(* CODESYS project Cowbell_Tracy_rev_2.project

Project tree, tasks and I/O mapping:
  Device : PAC320-CXX2X-XX, Parker Hannifin, order no. PAC320-CXX2X-XX, version 3.5.5.20
    application Application
      libraries: Util, 3.5.1.0 (System); CAA Types Extern, 3.5.5.0 (CAA Technical Workgroup); SysTypes Interfaces, * (System); CmpIecTask, 3.5.5.0 (System); SysFile, 3.5.5.0 (System); CmpErrors Interfaces, * (System); Unit Conversion Interfaces, * (Intern); SysTime, 3.5.5.0 (System)
      task EtherCAT_Master (externalevent, external event EVENT_ECM_DC, priority 0) calls EtherCAT_Master.EtherCAT_Task [EtherCAT_Master.EtherCAT_Task], DC_Monitor, RunLights, Rungs_First_500, Rungs_Second_500, RunMotion_All, Recovery, LogHiCycleCount
      task Slow_Task (cyclic, interval t#150ms, priority 20) calls PLC_PRG_1, Run_FileCopy, LogData
      global variables GVL
      global variables PersistentVars
      SymbolConfiguration
    SoftMotion General Axis Pool
      ZZ : SM_Drive_Virtual, 3S - Smart Software Solutions GmbH, order no. 1805, version 3.5.5.0
          settings: fRampJerk = 1e7
      A : SM_Drive_Virtual, 3S - Smart Software Solutions GmbH, order no. 1805, version 3.5.5.0
          settings: fRampJerk = 1e7
    EtherCAT_Master : PAC320 EtherCAT Master, Parker Hannifin, order no. PAC320-XXXXX-XX, version 3.5.5.0
        settings: MasterCycleTime = 1000
      Accelnet : Accelnet EtherCAT Drive (CoE) SoftMotion, Copley Controls Corp., version 3.5.5.0
          settings: EnableExpertSettings = True; StationAlias = 16; Optional = True; DC sync0 cycletime = 500; DC sync0 factor = 'x 1'; DC sync0 shift time = 0; DC sync1 cycletime = 500; DC sync1 factor = 'x 1'; DC sync1 shift time = 0; DCSetting = -1
          unmapped channels: Control word, Modes of operation, Target Position, Status word, Modes of operation display, Actual position
        Y : SM_Drive_ETC_Copley, 3S - Smart Software Solutions GmbH, order no. 0, version 3.5.5.0
            settings: AddressOffset_8010 = 20; BitOffset_8010 = 0; BitLength_8010 = 16; Address_8010 = '%QW10'; Type_8010 = 'UINT'; AddressPointer_8010 = ADR(%QW10); AddressOffset_8020 = 22; BitOffset_8020 = 0; BitLength_8020 = 8; Address_8020 = '%QB22'; Type_8020 = 'USINT'; AddressPointer_8020 = ADR(%QB22); AddressOffset_8030 = 24; BitOffset_8030 = 0; BitLength_8030 = 32; Address_8030 = '%QD6'; Type_8030 = 'DINT'; AddressPointer_8030 = ADR(%QD6); AddressOffset_8040 = 16#FFFFFFFF; BitOffset_8040 = 0; BitLength_8040 = 0; Address_8040 = ''; Type_8040 = ''; AddressPointer_8040 = 0; AddressOffset_8050 = 16#FFFFFFFF; BitOffset_8050 = 0; BitLength_8050 = 0; Address_8050 = ''; Type_8050 = ''; AddressPointer_8050 = 0; AdrOffset_8060 = 16#FFFFFFFF; BitOffset_8060 = 0; BitLength_8060 = 0; Address_8060 = ''; Type_8060 = ''; AddressPointer_8060 = 0; AdrOffset_8070 = 16#FFFFFFFF; BitOffset_8070 = 0; BitLength_8070 = 0; Address_8070 = '';
              Type_8070 = ''; AddressPointer_8070 = 0; AddressOffset_8510 = 24; BitOffset_8510 = 0; BitLength_8510 = 16; Address_8510 = '%IW12'; Type_8510 = 'UINT'; AddressPointer_8510 = ADR(%IW12); AddressOffset_8520 = 26; BitOffset_8520 = 0; BitLength_8520 = 8; Address_8520 = '%IB26'; Type_8520 = 'USINT'; AddressPointer_8520 = ADR(%IB26); AddressOffset_8530 = 28; BitOffset_8530 = 0; BitLength_8530 = 32; Address_8530 = '%ID7'; Type_8530 = 'DINT'; AddressPointer_8530 = ADR(%ID7); AddressOffset_8540 = 16#FFFFFFFF; BitOffset_8540 = 0; BitLength_8540 = 0; Address_8540 = ''; Type_8540 = ''; AddressPointer_8540 = 0; AddressOffset_8550 = 16#FFFFFFFF; BitOffset_8550 = 0; BitLength_8550 = 0; Address_8550 = ''; Type_8550 = ''; AddressPointer_8550 = 0
      Xenus_Plus_XEL : Xenus Plus EtherCAT Drive (CoE), Copley Controls, version Revision=16#00010003
          settings: EnableExpertSettings = True; Watchdog register 0400 = 2498; Watchdog register 0410 = 1000; Watchdog register 0420 = 1000; StationAlias = 17; DC sync0 cycletime = 1000; DC enable = 1; DC sync0 enable = 1; DC sync0 factor = 'x 1'; DC sync0 shift time = 0; DC sync1 cycletime = 1000; DC sync1 factor = 'x 1'; DC sync1 shift time = 0; DCSetting = 0; DC cyclic unit control = 48
          unmapped channels: Control word, Profile target position, Velocity offset, Torque offset, Status word, Actual motor position, Position loop error., Actual motor velocity, Torque actual value
        X : SM_Drive_ETC_GenericDSP402, 3S - Smart Software Solutions GmbH, order no. 0, version 3.5.5.0
            settings: dwRatioTechUnitsDenom = 4000; fPositionPeriod = 1; fRampJerk = 1e7; fSWLimitDeceleration = 0.0; fSWErrorMaxDistance = 0.0; ScalingIncs = 4000; AdrOffset_8010 = 4; BitOffset_8010 = 0; BitLength_8010 = 16; Address_8010 = '%QW2'; Type_8010 = 'UINT'; AddressPointer_8010 = ADR(%QW2); AdrOffset_8020 = 8; BitOffset_8020 = 0; BitLength_8020 = 32; Address_8020 = '%QD2'; Type_8020 = 'DINT'; AddressPointer_8020 = ADR(%QD2); AdrOffset_8030 = 16#FFFFFFFF; BitOffset_8030 = 0; BitLength_8030 = 0; Address_8030 = ''; Type_8030 = ''; AddressPointer_8030 = 0; AdrOffset_8040 = 16#FFFFFFFF; BitOffset_8040 = 0; BitLength_8040 = 0; Address_8040 = ''; Type_8040 = ''; AddressPointer_8040 = 0; AdrOffset_8050 = 16#FFFFFFFF; BitOffset_8050 = 0; BitLength_8050 = 0; Address_8050 = ''; Type_8050 = ''; AddressPointer_8050 = 0; AdrOffset_8060 = 16#FFFFFFFF; BitOffset_8060 = 0; BitLength_8060 = 0; Address_8060 = '';
              Type_8060 = ''; AddressPointer_8060 = 0; AdrOffset_8070 = 12; BitOffset_8070 = 0; BitLength_8070 = 32; Address_8070 = '%QD3'; Type_8070 = 'DINT'; AddressPointer_8070 = ADR(%QD3); AdrOffset_8080 = 16; BitOffset_8080 = 0; BitLength_8080 = 16; Address_8080 = '%QW8'; Type_8080 = 'INT'; AddressPointer_8080 = ADR(%QW8); AdrOffset_8510 = 4; BitOffset_8510 = 0; BitLength_8510 = 16; Address_8510 = '%IW2'; Type_8510 = 'UINT'; AddressPointer_8510 = ADR(%IW2); AdrOffset_8520 = 8; BitOffset_8520 = 0; BitLength_8520 = 32; Address_8520 = '%ID2'; Type_8520 = 'DINT'; AddressPointer_8520 = ADR(%ID2); AdrOffset_8530 = 16; BitOffset_8530 = 0; BitLength_8530 = 32; Address_8530 = '%ID4'; Type_8530 = 'DINT'; AddressPointer_8530 = ADR(%ID4); AdrOffset_8540 = 20; BitOffset_8540 = 0; BitLength_8540 = 16; Address_8540 = '%IW10'; Type_8540 = 'INT'; AddressPointer_8540 = ADR(%IW10); AdrOffset_8550 = 16#FFFFFFFF; BitOffset_8550 = 0;
              BitLength_8550 = 0; Address_8550 = ''; Type_8550 = ''; AddressPointer_8550 = 0; AdrOffset_8560 = 16#FFFFFFFF; BitOffset_8560 = 0; BitLength_8560 = 0; Address_8560 = ''; Type_8560 = ''; AddressPointer_8560 = 0; AdrOffset_8570 = 16#FFFFFFFF; BitOffset_8570 = 0; BitLength_8570 = 0; Address_8570 = ''; Type_8570 = ''; AddressPointer_8570 = 0; AdrOffset_8580 = 16#FFFFFFFF; BitOffset_8580 = 0; BitLength_8580 = 0; Address_8580 = ''; Type_8580 = ''; AddressPointer_8580 = 0; AdrOffset_8590 = 16#FFFFFFFF; BitOffset_8590 = 0; BitLength_8590 = 0; Address_8590 = ''; Type_8590 = ''; AddressPointer_8590 = 0; AdrOffset_8600 = 16#FFFFFFFF; BitOffset_8600 = 0; BitLength_8600 = 0; Address_8600 = ''; Type_8600 = ''; AddressPointer_8600 = 0; AdrOffset_8600 = 16#FFFFFFFF; BitOffset_8600 = 0; BitLength_8600 = 0; Address_8610 = ''; Type_8610 = ''; AddressPointer_8610 = 0
      PAC320_BusCoupler : PAC320 BusCoupler, Parker Hannifin, version Revision=16#00000001
          settings: EnableExpertSettings = True; StationAlias = 1; DC sync0 cycletime = 500; DC enable = 1; DC sync0 enable = 1; DC sync0 factor = 'x 1'; DC sync0 shift time = 0; DC sync1 cycletime = 500; DC sync1 enable = 0; DC sync1 factor = 'x 1'; DC sync1 shift time = 0
        PACIO_DI16_DO16 : DI16/DO16 1ms 0.5A (PACIO-450-03), Parker Hannifin, version Revision=16#00000001
            settings: StationAlias = 0; DC sync0 cycletime = 500; DC sync1 cycletime = 500
            output A_Output00 : BIT  // DigitalOutput0
            output A_Output01 : BIT  // DigitalOutput1
            output A_Output02 : BIT  // DigitalOutput2
            output A_Output03 : BIT  // DigitalOutput3
            output A_Output04 : BIT  // DigitalOutput4
            output A_Output05 : BIT  // DigitalOutput5
            output A_Output06 : BIT  // DigitalOutput6
            output A_Output07 : BIT  // DigitalOutput7
            output A_Output08 : BIT  // DigitalOutput8
            output A_Output09 : BIT  // DigitalOutput9
            output A_Output10 : BIT  // DigitalOutput10
            output A_Output11 : BIT  // DigitalOutput11
            output A_Output12 : BIT  // DigitalOutput12
            output A_Output13 : BIT  // DigitalOutput13
            output A_Output14 : BIT  // DigitalOutput14
            output A_Output15 : BIT  // DigitalOutput15
            input  A_Input00 : BIT  // DigitalInput0
            input  A_Input01 : BIT  // DigitalInput1
            input  A_Input02 : BIT  // DigitalInput2
            input  A_Input03 : BIT  // DigitalInput3
            input  A_Input04 : BIT  // DigitalInput4
            input  A_Input05 : BIT  // DigitalInput5
            input  A_Input06 : BIT  // DigitalInput6
            input  A_Input07 : BIT  // DigitalInput7
            input  In_Power : BIT  // DigitalInput8
            input  In_Reset : BIT  // DigitalInput9
            input  In_Neg : BIT  // DigitalInput10
            input  In_Pos : BIT  // DigitalInput11
            input  In_Zero : BIT  // DigitalInput12
            input  In_Start : BIT  // DigitalInput13
            input  In_Stop : BIT  // DigitalInput14
            input  In_Cycle : BIT  // DigitalInput15
        PACIO_DI16_DO16_1 : DI16/DO16 1ms 0.5A (PACIO-450-03), Parker Hannifin, version Revision=16#00000001
            settings: StationAlias = 0; DC sync0 cycletime = 500; DC sync1 cycletime = 500
            output B_Output00 : BIT  // DigitalOutput0
            output B_Output01 : BIT  // DigitalOutput1
            output B_Output02 : BIT  // DigitalOutput2
            output B_Output03 : BIT  // DigitalOutput3
            output B_Output04 : BIT  // DigitalOutput4
            output B_Output05 : BIT  // DigitalOutput5
            output B_Output06 : BIT  // DigitalOutput6
            output B_Output07 : BIT  // DigitalOutput7
            output B_Output08 : BIT  // DigitalOutput8
            output B_Output09 : BIT  // DigitalOutput9
            output B_Output10 : BIT  // DigitalOutput10
            output B_Output11 : BIT  // DigitalOutput11
            output B_Output12 : BIT  // DigitalOutput12
            output B_Output13 : BIT  // DigitalOutput13
            output B_Output14 : BIT  // DigitalOutput14
            output B_Output15 : BIT  // DigitalOutput15
            input  B_Input00 : BIT  // DigitalInput0
            input  B_Input01 : BIT  // DigitalInput1
            input  B_Input02 : BIT  // DigitalInput2
            input  B_Input03 : BIT  // DigitalInput3
            input  B_Input04 : BIT  // DigitalInput4
            input  B_Input05 : BIT  // DigitalInput5
            input  B_Input06 : BIT  // DigitalInput6
            input  B_Input07 : BIT  // DigitalInput7
            input  B_Input08 : BIT  // DigitalInput8
            input  B_Input09 : BIT  // DigitalInput9
            input  B_Input10 : BIT  // DigitalInput10
            input  B_Input11 : BIT  // DigitalInput11
            input  B_Input12 : BIT  // DigitalInput12
            input  B_Input13 : BIT  // DigitalInput13
            input  B_Input14 : BIT  // DigitalInput14
            input  B_Input15 : BIT  // DigitalInput15
      Compax3_EtherCat_DS402_CoE : C3SxxxVxFxxI31T11Mxx_OpMode08 V2.05 SoftMotion, Parker Hannifin, version 3.5.5.0
          settings: EnableExpertSettings = True; StationAlias = 1006; Optional = True; DC sync0 cycletime = 4000; DC enable = 1; DC sync0 enable = 1; DC sync0 factor = 'x 4'; DC sync0 shift time = 0; DC sync1 cycletime = 4000; DC sync1 enable = 0; DC sync1 shift time = 0
          unmapped channels: Controlword, Target Position, Dig.Outputs, ModeofOperation, Statusword, Actual Position, Dig.Inputs, ModeOfOperationDisplay
        Z : SM_Drive_ETC_PARKER, 3S - Smart Software Solutions GmbH, order no. 0, version 3.5.5.0
            settings: dwRatioTechUnitsDenom = 4096; ScalingIncs = 4096; AdrOffset_8010 = 28; BitOffset_8010 = 0; BitLength_8010 = 16; Address_8010 = '%QW14'; Type_8010 = 'UINT'; AddressPointer_8010 = ADR(%QW14); AdrOffset_8020 = 32; BitOffset_8020 = 0; BitLength_8020 = 32; Address_8020 = '%QD8'; Type_8020 = 'DINT'; AddressPointer_8020 = ADR(%QD8); AdrOffset_8030 = 38; BitOffset_8030 = 0; BitLength_8030 = 16; Address_8030 = '%QW19'; Type_8030 = 'INT'; AddressPointer_8030 = ADR(%QW19); AdrOffset_8040 = 36; BitOffset_8040 = 0; BitLength_8040 = 16; Address_8040 = '%QW18'; Type_8040 = 'UINT'; AddressPointer_8040 = ADR(%QW18); AdrOffset_8510 = 32; BitOffset_8510 = 0; BitLength_8510 = 16; Address_8510 = '%IW16'; Type_8510 = 'UINT'; AddressPointer_8510 = ADR(%IW16); AdrOffset_8520 = 16#FFFFFFFF; BitOffset_8520 = 0; BitLength_8520 = 0; Address_8520 = ''; Type_8520 = ''; AddressPointer_8520 = 0; AdrOffset_8530 = 42; BitOffset_8530 = 0;
              BitLength_8530 = 16; Address_8530 = '%IW21'; Type_8530 = 'INT'; AddressPointer_8530 = ADR(%IW21); AdrOffset_8540 = 40; BitOffset_8540 = 0; BitLength_8540 = 16; Address_8540 = '%IW20'; Type_8540 = 'UINT'; AddressPointer_8540 = ADR(%IW20); AdrOffset_8550 = 36; BitOffset_8550 = 0; BitLength_8550 = 32; Address_8550 = '%ID9'; Type_8550 = 'DINT'; AddressPointer_8550 = ADR(%ID9)
    Ethernet : Ethernet, 3S - Smart Software Solutions GmbH, version 3.4.2.0
      ModbusTCP_Slave_Device : ModbusTCP Slave Device, 3S - Smart Software Solutions GmbH, version 3.5.5.0
          input  Application.DC_Monitor.HMI_ResetCounter : WORD  // Inputs.Inputs
          output Application.DC_Monitor.Captured_CycleTime_Avg : WORD  // Outputs.Outputs
          output Application.DC_Monitor.Captured_CycleTime_Max : WORD  // Outputs.Outputs
          output Application.DC_Monitor.Captured_CycleTime_Min : WORD  // Outputs.Outputs
          output Application.DC_Monitor.Captured_MaxTotalSyncBufferAvg : WORD  // Outputs.Outputs
          output Application.DC_Monitor.CycleTime_Avg : WORD  // Outputs.Outputs
          output Application.DC_Monitor.CycleTime_Max : WORD  // Outputs.Outputs
          output Application.DC_Monitor.CycleTime_Min : WORD  // Outputs.Outputs
          output Application.DC_Monitor.CycleTime_Count : WORD  // Outputs.Outputs
          output Application.DC_Monitor.CycleTime_Last : WORD  // Outputs.Outputs
          output Application.MaxTotalSyncBufferAvg : WORD  // Outputs.Outputs
          output Application.DC_Monitor.TotalSyncBufferAvg : WORD  // Outputs.Outputs
          output Application.RunLights.iCycle : WORD  // Outputs.Outputs
          output Application.RunMotion_All.DoMotion_X.HMI_ActualPosition : WORD  // Outputs.Outputs
          output Application.DC_Monitor.HMI_DC_InSync : WORD  // Outputs.Outputs
          output Application.dcWindow : WORD  // Outputs.Outputs
          output Application.gSyncErrors : WORD  // Outputs.Outputs
          unmapped channels: Inputs, Outputs
  program PLC_PRG [CFC]
  program RunSDO_AOut [ST]
  function block GetSDO_AOut [CFC]
  function block GetSDO [CFC]
  function block SetOutputs [ST]
  function block GetInputs [ST]
  function block SetAnalogVoltage [ST]
  function VOLTS_to_UINT [ST]
  function UINT_to_VOLTS [ST]
  program RunSDO [ST]
  function block GetAnalogVoltage [ST]
  function block InitSDO [ST]
  function block ConfigAnalogVoltage [ST]
  program RunMotion_old [ST]
  function block IO_AxisControl [CFC]
  program POU_X [CFC]
  function block SetSDO_AOut [CFC]
  function block InitSDO_Y [ST]
  program RunMotion_Y_old [ST]
  program RunSDO_Y [ST]
  program RunSDO_AOut_Y [ST]
  function block GetSDO_Y [CFC]
  function block GetSDO_AOut_Y [CFC]
  function block SetSDO_AOut_Y [CFC]
  function GetHeaderString [ST]
  program DC_Monitor [ST]
  program RunLights [ST]
  program RunMotion_Z_old [ST]
  program RunMotion_A [ST]
  function block MotionFB [ST]
  program Recovery [ST]
  program RunMotion_All [ST]
  function GetLogMsgString [ST]
  program LogHiCycleCount [ST]
  function GetTimeStampString [ST]
  text list GlobalTextList
  function AllTaskInfo [ST]
  function CurrentTaskInfo [ST]
  function ResetTaskInfo [ST]
  program Rungs_First_500 [LD]
  program Rungs_Second_500 [LD]
  program RunMotion [ST]
  program RunMotion_Y [ST]
  program RunMotion_Z [ST]
  function block Test_FileCopy [ST]
  program Run_FileCopy [CFC]
  program PLC_PRG_1 [ST]
  program LogData [ST]
  function My_FLOAT_TO_STRING [ST]
  function GetTimeStampString_1 [ST]
*)

// Device/Application/GVL
VAR_GLOBAL
	g_PosDistance:REAL := 20.0;
	g_NegDistance:REAL := -20.0;
	g_Vel:REAL := 5.0;
	g_Acc:REAL := 10.0;
	//In_Power : BOOL ;
	//In_Reset : BOOL;
	//In_Pos : BOOL;
	//In_Neg : BOOL;
	//In_Stop : BOOL;
	//In_Zero : BOOL;
	g_MoveDwellPos : BOOL := FALSE;
	g_MoveDwellNeg : BOOL := FALSE;
	g_MoveDwellPos_Y : BOOL := FALSE;
	g_MoveDwellNeg_Y : BOOL := FALSE;
	g_MoveDwellPos_Z : BOOL := FALSE;
	g_MoveDwellNeg_Z : BOOL := FALSE;
	g_MoveDwellPos_A : BOOL := FALSE;
	g_MoveDwellNeg_A : BOOL := FALSE;
	g_GotSDO_PostionPos : BOOL;
	g_GotSDO_PostionNeg : BOOL;
	g_GotSDO_Y_PostionPos : BOOL;
	g_GotSDO_Y_PostionNeg : BOOL;
	DC_InSync: BOOL;
	g_FirstSync: BOOL;
	g_LostSync: BOOL;
	
	
	//ScanTimeMax: DINT;
	//ScanTimeMin: DINT;
	//dcWindow: WORD := 50;

	//MaxScanTime: DINT;
	//MaxSyncTime: DINT;
	//MinSyncTime: DINT;
	//MaxTotalSyncBufferAvg: DINT;
	MyArray: ARRAY[0..9, 0..9] OF REAL;
END_VAR

// Device/Application/PersistentVars
VAR_GLOBAL PERSISTENT RETAIN
	ScanTimeMax: DINT;
	ScanTimeMin: DINT;
	dcWindow: WORD ;

	MaxScanTime: DINT;
	MaxSyncTime: DINT;
	MinSyncTime: DINT;
	MaxTotalSyncBufferAvg: DINT;

	gSyncErrors: DINT;
END_VAR

// DC_Monitor
PROGRAM DC_Monitor
VAR
	TurnON_LED_A: BOOL;
	TurnON_LED_B: BOOL;
	m_master: INT;
	ResetLED: BOOL := FALSE;
	iLoopCount: UINT;
	CurrentScanTime: DINT;
	CurrentSyncTime: DINT;
	SyncBufferMax: DINT;
	TotalSyncBuffer: DINT;
	TotalSyncBufferAvg: DINT;
	tTask 			: Task_Info2; (* Information about the task *)
	pTask2			: POINTER  TO Task_Info2;
	aIecTasks 		: ARRAY[1..20] OF Task_Info2; (* Information about all tasks *)
	sAppName		: STRING := 'Application';
	
	hCurrentTask	: RTS_IEC_HANDLE; (* Current task *)
	hSlowTask		: RTS_IEC_HANDLE; (* The slower task handle*)
	hReloaded 		: RTS_IEC_HANDLE; (* Reloaded task *)
	Result			: RTS_IEC_RESULT; (* Result Code *)
	ResetStats : BOOL;
	ResetResult		: RTS_IEC_RESULT; (* Reset Result Code *)
	DoReset : BOOL := FALSE;
	DoAutoReset : BOOL := FALSE;
	Capture_Done : BOOL := FALSE;
	Captured_CycleTime_Avg : DWORD := 0;
	Captured_CycleTime_Max : DWORD := 0;
	Captured_CycleTime_Min : DWORD := 0;
	Captured_MaxTotalSyncBufferAvg : DINT := 0;
	
	
	CyclesIn5min: UDINT;
	CycleTime_Avg: DWORD;
	CycleTime_Max: DWORD;
	CycleTime_Min: DWORD;
	CycleTime_Last: DWORD;
	CycleTime_Count: DWORD;
	
	HMI_ResetCounter : WORD;
	HMI_DC_InSync : WORD;
	
END_VAR

EtherCAT_Master();
dcWindow := EtherCAT_Master.DCInSyncWindow;
//ScanTimeMax := EtherCAT_Master.m_master.m_diMaxSyncTime;
//ScanTimeMin := EtherCAT_Master.m_master.m_diMinSyncTime;
DC_InSync := EtherCAT_Master.xDistributedClockInSync;
(* Current task information, some of these information can be find in the Task Configuration under the monitor tab.*)
tTask := CurrentTaskInfo();
	CycleTime_Avg := tTask.dwAverageCycleTime;
	CycleTime_Max := tTask.dwMaxCycleTime;
	CycleTime_Min := tTask.dwMinCycleTime;
	CycleTime_Last := tTask.dwCycleTime; 
	CycleTime_Count := tTask.dwCycleCount / 2000;
	DoReset := HMI_ResetCounter.0;
	HMI_DC_InSync.0 := DC_InSync;
	

IF DoReset OR DoAutoReset THEN
	ResetResult := ResetTaskInfo();
	MaxTotalSyncBufferAvg := 0;
	Capture_Done := FALSE;
	Captured_CycleTime_Avg := 0;
	Captured_CycleTime_Max := 0;
	Captured_CycleTime_Min := 0;
	Captured_MaxTotalSyncBufferAvg := 0;
	DoReset := FALSE;
	DoAutoReset := FALSE;
END_IF;


TotalSyncBuffer := 0;
FOR iLoopCount:=0 TO ETHERCAT_PLL_BUFFER - 1 DO
	CurrentScanTime := ABS(EtherCAT_Master.m_master.m_diSyncBuffer[iLoopCount]);
    TotalSyncBuffer := TotalSyncBuffer + CurrentScanTime;
	IF(CurrentScanTime > ScanTimeMax) THEN
		SyncBufferMax := CurrentScanTime;
	END_IF
END_FOR

TotalSyncBufferAvg := TotalSyncBuffer/ETHERCAT_PLL_BUFFER;
IF(TotalSyncBufferAvg > MaxTotalSyncBufferAvg AND g_FirstSync) THEN
	MaxTotalSyncBufferAvg := TotalSyncBufferAvg;
END_IF

iLoopCount := 0;
FOR iLoopCount:=0 TO 49 DO
	CurrentScanTime := EtherCAT_Master.m_master.m_diIntervallBuffer[iLoopCount]; 
	IF(CurrentScanTime > MaxScanTime) THEN
		MaxScanTime := CurrentScanTime;
	END_IF
END_FOR

(* Not Available without Debug
CurrentSyncTime := EtherCAT_Master.m_master.m_diMaxSyncTime;
IF(CurrentSyncTime > MaxSyncTime AND g_FirstSync) THEN
	MaxSyncTime := CurrentSyncTime;
END_IF

CurrentSyncTime := EtherCAT_Master.m_master.m_diMinSyncTime;
IF(CurrentSyncTime < MinSyncTime AND g_FirstSync) THEN
	MinSyncTime := CurrentSyncTime;
END_IF
*)
CyclesIn5min := (5 * 60 * 1000000) / tTask.dwInterval; //Need to get the EtherCAT CycleTime
IF (tTask.dwIECCycleCount > CyclesIn5min) AND Capture_Done = FALSE THEN
	Captured_CycleTime_Avg := tTask.dwAverageCycleTime;
	Captured_CycleTime_Max := tTask.dwMaxCycleTime;
	Captured_CycleTime_Min := tTask.dwMinCycleTime;
	Captured_MaxTotalSyncBufferAvg := MaxTotalSyncBufferAvg;

	Capture_Done := TRUE;
	
END_IF



IF (ResetLED) THEN
	//CmpToggleLED.SetLED_A(FALSE);
	g_LostSync := FALSE;
	MaxSyncTime := 0;
	MinSyncTime := 0;
	ResetLED := FALSE;
END_IF

IF NOT EtherCAT_Master.xDistributedClockInSync THEN
	//CmpToggleLED.SetLED_A(TRUE);
	g_LostSync := TRUE;
END_IF

IF EtherCAT_Master.xDistributedClockInSync AND NOT g_FirstSync THEN
	g_FirstSync := TRUE;	
	g_LostSync := FALSE;
	DoAutoReset := TRUE;
END_IF

END_PROGRAM

// CurrentTaskInfo
FUNCTION CurrentTaskInfo : Task_Info2
VAR_INPUT
END_VAR

VAR
	Result 	: RTS_IEC_RESULT;
	hIecTask: RTS_IEC_HANDLE;
END_VAR

(* Task information about the current task are returned *)
hIecTask := IecTaskGetCurrent(pResult:=ADR(Result));
IF hIecTask <> RTS_INVALID_HANDLE AND Result = 0 THEN
	CurrentTaskInfo := IecTaskGetInfo3(hIecTask:=hIecTask, pResult:=ADR(Result))^;
END_IF

END_FUNCTION

// ResetTaskInfo
FUNCTION ResetTaskInfo : RTS_IEC_RESULT
VAR_INPUT
END_VAR
VAR
	Result 	: RTS_IEC_RESULT;
	PResult 	: RTS_IEC_RESULT;
	Handle: RTS_IEC_HANDLE;
END_VAR

(* Task information about the current task are returned *)
Handle := IecTaskGetCurrent(pResult:=ADR(PResult));
IF Handle <> RTS_INVALID_HANDLE AND PResult = 0 THEN
	ResetTaskInfo := IecTaskResetStatistics(hIecTask:=Handle);
END_IF

END_FUNCTION

// RunLights
PROGRAM RunLights
VAR
	iStatus: INT := -1;
	iCycle: INT;
	iCycleMin: INT := 0;
	iCycleMax: INT := 9;
	DoOutputs : SetOutputs;
	DoInputs : GetInputs;
	TimerON : TON;
	TimerON2 : TON;
	tWait: TIME := T#0.25S;
	tWait2: TIME := T#0.25S;
	//tWait: TIME := T#1S;
	//tWait2: TIME := T#4S;
	iIncrement: INT := 1;
	uiExpectedValue: UINT;
	uiActualValue: UINT;
END_VAR

(*IF PACIO_DI16_DO16.wState <> ETC_SLAVE_STATE.ETC_SLAVE_OPERATIONAL THEN
	RETURN;
END_IF
*)


CASE iStatus OF
	
-1: //Wait Time
	//TimerON(PT:=tWaitPowerup, IN:=TRUE);
	IF EtherCAT_Master.xConfigFinished THEN
		//TimerON(IN:=FALSE,PT:=T#0S);
		iStatus:=iStatus + 1;
	END_IF
	
0: //Set Outputs
	uiExpectedValue := LREAL_TO_UINT(EXPT(2,iCycle));
	DoOutputs(OutputValue := uiExpectedValue,Execute:=TRUE);
	IF DoOutputs.Done THEN
		iCycle:=iCycle + iIncrement;
		IF iCycle = iCycleMax THEN
			iIncrement:=-1;
		END_IF;
		IF iCycle = iCycleMin THEN
			iIncrement:= 1;
		END_IF;
		iStatus:=1;	
	END_IF;
1: //Wait Time
	TimerON(PT:=tWait, IN:=TRUE);
	IF TimerON.Q=TRUE THEN
		TimerON(IN:=FALSE,PT:=T#0S);
		iStatus:=2;
	END_IF
2: //Check Inputs
	DoInputs(Execute:=TRUE );
	IF DoInputs.Done = TRUE THEN
		uiActualValue:=DoInputs.InputValue;
		IF uiActualValue = uiExpectedValue THEN
			A_Output00 := FALSE;
		ELSE 
			A_Output00 :=TRUE;	
		END_IF
		DoOutputs(Execute:=FALSE);
		DoInputs(Execute:=FALSE);
		iStatus:=3;	
		
	END_IF
3: //Wait Time
	TimerON2(PT:=tWait2, IN:=TRUE);
	IF TimerON2.Q=TRUE THEN
		TimerON2(IN:=FALSE,PT:=T#0S);
		iStatus:=0;
	END_IF
	

END_CASE;

END_PROGRAM

// SetOutputs
FUNCTION_BLOCK SetOutputs
VAR_INPUT
	Execute: BOOL;
	OutputValue: UINT;
END_VAR
VAR_OUTPUT
	Busy: BOOL;
	Done: BOOL;
END_VAR
VAR
	iStatus: INT := 0;
(*	Output00: BOOL;
	Output01: BOOL;
	Output02: BOOL;
	Output03: BOOL;
	Output04: BOOL;
	Output05: BOOL;
	Output06: BOOL;
	Output07: BOOL;
	Output08: BOOL;
	Output09: BOOL;
	Output10: BOOL;
	Output11: BOOL;
	Output12: BOOL;
	Output13: BOOL;
	Output14: BOOL;
	Output15: BOOL;
*)
END_VAR

CASE iStatus OF
	
0: //Waiting for Execute = True
	IF Execute = TRUE THEN
		Busy:=TRUE;
		Done:=FALSE;
		iStatus := iStatus + 1;
		
	END_IF;

1:
	A_Output15:= OutputValue.0;
	A_Output14:= OutputValue.1;
	A_Output13:= OutputValue.2;
	A_Output12:= OutputValue.3;
	A_Output11:= OutputValue.4;
	A_Output10:= OutputValue.5;
	A_Output09:= OutputValue.6;
	A_Output08:= OutputValue.7;
	A_Output07:= OutputValue.8;
	A_Output06:= OutputValue.9;
	A_Output05:= OutputValue.10;
	A_Output04:= OutputValue.11;
	A_Output03:= OutputValue.12;
	A_Output02:= OutputValue.13;
	A_Output01:= OutputValue.14;
	A_Output00:= OutputValue.15;	
(*
	
	B_Output15:= OutputValue.0;
	B_Output14:= OutputValue.1;
	B_Output13:= OutputValue.2;
	B_Output12:= OutputValue.3;
	B_Output11:= OutputValue.4;
	B_Output10:= OutputValue.5;
	B_Output09:= OutputValue.6;
	B_Output08:= OutputValue.7;
	B_Output07:= OutputValue.8;
	B_Output06:= OutputValue.9;
	B_Output05:= OutputValue.10;
	B_Output04:= OutputValue.11;
	B_Output03:= OutputValue.12;
	B_Output02:= OutputValue.13;
	B_Output01:= OutputValue.14;
	B_Output00:= OutputValue.15;
*)
	Busy:=FALSE;
	Done:=TRUE;
	iStatus := iStatus + 1;

2://Waiting for Execute = False
	IF Execute = FALSE THEN
		iStatus := 0;
	END_IF;

END_CASE;

END_FUNCTION_BLOCK

// GetInputs
FUNCTION_BLOCK GetInputs
VAR_INPUT
	Execute: BOOL;
	
END_VAR
VAR_OUTPUT
	Busy: BOOL;
	Done: BOOL;
	InputValue: UINT;
END_VAR
VAR
	iStatus: INT := 0;
(*	Input00: BOOL;
	Input01: BOOL;
	Input02: BOOL;
	Input03: BOOL;
	Input04: BOOL;
	Input05: BOOL;
	Input06: BOOL;
	Input07: BOOL;
	Input08: BOOL;
	Input09: BOOL;
	Input10: BOOL;
	Input11: BOOL;
	Input12: BOOL;
	Input13: BOOL;
	Input14: BOOL;
	Input15: BOOL;
*)
END_VAR

CASE iStatus OF
	
0: //Waiting for Execute = True
	IF Execute = TRUE THEN
		Busy:=TRUE;
		Done:=FALSE;
		iStatus := iStatus + 1;
		
	END_IF;

1:
	InputValue.0:= In_Cycle;
	InputValue.1:= In_Stop;
	InputValue.2:= In_Start;
	InputValue.3:= In_Zero;
	InputValue.4:= In_Pos;
	InputValue.5:= In_Neg;
	InputValue.6:= In_Reset;
	InputValue.7:= In_Power;
	InputValue.8:= A_Input07;
	InputValue.9:= A_Input06;
	InputValue.10:= In_Neg;
	InputValue.11:= In_Pos;
	InputValue.12:= In_Zero;
	InputValue.13:= In_Start; 
	InputValue.14:= In_Stop; 
	InputValue.15:= In_Cycle; 
	Busy:=FALSE;
	Done:=TRUE;
	iStatus := iStatus + 1;

2://Waiting for Execute = False
	IF Execute = FALSE THEN
		iStatus := 0;
	END_IF;

END_CASE;

END_FUNCTION_BLOCK

// Rungs_First_500
PROGRAM Rungs_First_500
VAR
VAR004 :INT := 96;
VAR000 :INT := 96;
BContactBit0000	:BOOL;
BContactBit0001	:BOOL;
BContactBit0002	:BOOL;
BContactBit0003	:BOOL;
BContactBit0004	:BOOL;
BContactBit0005	:BOOL;
BContactBit0006	:BOOL;
BContactBit0007	:BOOL;
BContactBit0008	:BOOL;
BContactBit0009	:BOOL;
BContactBit0010	:BOOL;
BContactBit0011	:BOOL;
BContactBit0012	:BOOL;
BContactBit0013	:BOOL;
BContactBit0014	:BOOL;
BContactBit0015	:BOOL;
BContactBit0016	:BOOL;
BContactBit0017	:BOOL;
BContactBit0018	:BOOL;
BContactBit0019	:BOOL;
BContactBit0020	:BOOL;
BContactBit0021	:BOOL;
BContactBit0022	:BOOL;
BContactBit0023	:BOOL;
BContactBit0024	:BOOL;
BContactBit0025	:BOOL;
BContactBit0026	:BOOL;
BContactBit0027	:BOOL;
BContactBit0028	:BOOL;
BContactBit0029	:BOOL;
BContactBit0030	:BOOL;
BContactBit0031	:BOOL;
BContactBit0032	:BOOL;
BContactBit0033	:BOOL;
BContactBit0034	:BOOL;
BContactBit0035	:BOOL;
BContactBit0036	:BOOL;
BContactBit0037	:BOOL;
BContactBit0038	:BOOL;
BContactBit0039	:BOOL;
BContactBit0040	:BOOL;
BContactBit0041	:BOOL;
BContactBit0042	:BOOL;
BContactBit0043	:BOOL;
BContactBit0044	:BOOL;
BContactBit0045	:BOOL;
BContactBit0046	:BOOL;
BContactBit0047	:BOOL;
BContactBit0048	:BOOL;
BContactBit0049	:BOOL;
BContactBit0050	:BOOL;
BContactBit0051	:BOOL;
BContactBit0052	:BOOL;
BContactBit0053	:BOOL;
BContactBit0054	:BOOL;
BContactBit0055	:BOOL;
BContactBit0056	:BOOL;
BContactBit0057	:BOOL;
BContactBit0058	:BOOL;
BContactBit0059	:BOOL;
BContactBit0060	:BOOL;
BContactBit0061	:BOOL;
BContactBit0062	:BOOL;
BContactBit0063	:BOOL;
BContactBit0064	:BOOL;
BContactBit0065	:BOOL;
BContactBit0066	:BOOL;
BContactBit0067	:BOOL;
BContactBit0068	:BOOL;
BContactBit0069	:BOOL;
BContactBit0070	:BOOL;
BContactBit0071	:BOOL;
BContactBit0072	:BOOL;
BContactBit0073	:BOOL;
BContactBit0074	:BOOL;
BContactBit0075	:BOOL;
BContactBit0076	:BOOL;
BContactBit0077	:BOOL;
BContactBit0078	:BOOL;
BContactBit0079	:BOOL;
BContactBit0080	:BOOL;
BContactBit0081	:BOOL;
BContactBit0082	:BOOL;
BContactBit0083	:BOOL;
BContactBit0084	:BOOL;
BContactBit0085	:BOOL;
BContactBit0086	:BOOL;
BContactBit0087	:BOOL;
BContactBit0088	:BOOL;
BContactBit0089	:BOOL;
BContactBit0090	:BOOL;
BContactBit0091	:BOOL;
BContactBit0092	:BOOL;
BContactBit0093	:BOOL;
BContactBit0094	:BOOL;
BContactBit0095	:BOOL;
BContactBit0096	:BOOL;
BContactBit0097	:BOOL;
BContactBit0098	:BOOL;
BContactBit0099	:BOOL;
BContactBit0100	:BOOL;
BContactBit0101	:BOOL;
BContactBit0102	:BOOL;
BContactBit0103	:BOOL;
BContactBit0104	:BOOL;
BContactBit0105	:BOOL;
BContactBit0106	:BOOL;
BContactBit0107	:BOOL;
BContactBit0108	:BOOL;
BContactBit0109	:BOOL;
BContactBit0110	:BOOL;
BContactBit0111	:BOOL;
BContactBit0112	:BOOL;
BContactBit0113	:BOOL;
BContactBit0114	:BOOL;
BContactBit0115	:BOOL;
BContactBit0116	:BOOL;
BContactBit0117	:BOOL;
BContactBit0118	:BOOL;
BContactBit0119	:BOOL;
BContactBit0120	:BOOL;
BContactBit0121	:BOOL;
BContactBit0122	:BOOL;
BContactBit0123	:BOOL;
BContactBit0124	:BOOL;
BContactBit0125	:BOOL;
BContactBit0126	:BOOL;
BContactBit0127	:BOOL;
BContactBit0128	:BOOL;
BContactBit0129	:BOOL;
BContactBit0130	:BOOL;
BContactBit0131	:BOOL;
BContactBit0132	:BOOL;
BContactBit0133	:BOOL;
BContactBit0134	:BOOL;
BContactBit0135	:BOOL;
BContactBit0136	:BOOL;
BContactBit0137	:BOOL;
BContactBit0138	:BOOL;
BContactBit0139	:BOOL;
BContactBit0140	:BOOL;
BContactBit0141	:BOOL;
BContactBit0142	:BOOL;
BContactBit0143	:BOOL;
BContactBit0144	:BOOL;
BContactBit0145	:BOOL;
BContactBit0146	:BOOL;
BContactBit0147	:BOOL;
BContactBit0148	:BOOL;
BContactBit0149	:BOOL;
BContactBit0150	:BOOL;
BContactBit0151	:BOOL;
BContactBit0152	:BOOL;
BContactBit0153	:BOOL;
BContactBit0154	:BOOL;
BContactBit0155	:BOOL;
BContactBit0156	:BOOL;
BContactBit0157	:BOOL;
BContactBit0158	:BOOL;
BContactBit0159	:BOOL;
BContactBit0160	:BOOL;
BContactBit0161	:BOOL;
BContactBit0162	:BOOL;
BContactBit0163	:BOOL;
BContactBit0164	:BOOL;
BContactBit0165	:BOOL;
BContactBit0166	:BOOL;
BContactBit0167	:BOOL;
BContactBit0168	:BOOL;
BContactBit0169	:BOOL;
BContactBit0170	:BOOL;
BContactBit0171	:BOOL;
BContactBit0172	:BOOL;
BContactBit0173	:BOOL;
BContactBit0174	:BOOL;
BContactBit0175	:BOOL;
BContactBit0176	:BOOL;
BContactBit0177	:BOOL;
BContactBit0178	:BOOL;
BContactBit0179	:BOOL;
BContactBit0180	:BOOL;
BContactBit0181	:BOOL;
BContactBit0182	:BOOL;
BContactBit0183	:BOOL;
BContactBit0184	:BOOL;
BContactBit0185	:BOOL;
BContactBit0186	:BOOL;
BContactBit0187	:BOOL;
BContactBit0188	:BOOL;
BContactBit0189	:BOOL;
BContactBit0190	:BOOL;
BContactBit0191	:BOOL;
BContactBit0192	:BOOL;
BContactBit0193	:BOOL;
BContactBit0194	:BOOL;
BContactBit0195	:BOOL;
BContactBit0196	:BOOL;
BContactBit0197	:BOOL;
BContactBit0198	:BOOL;
BContactBit0199	:BOOL;
BContactBit0200	:BOOL;
BContactBit0201	:BOOL;
BContactBit0202	:BOOL;
BContactBit0203	:BOOL;
BContactBit0204	:BOOL;
BContactBit0205	:BOOL;
BContactBit0206	:BOOL;
BContactBit0207	:BOOL;
BContactBit0208	:BOOL;
BContactBit0209	:BOOL;
BContactBit0210	:BOOL;
BContactBit0211	:BOOL;
BContactBit0212	:BOOL;
BContactBit0213	:BOOL;
BContactBit0214	:BOOL;
BContactBit0215	:BOOL;
BContactBit0216	:BOOL;
BContactBit0217	:BOOL;
BContactBit0218	:BOOL;
BContactBit0219	:BOOL;
BContactBit0220	:BOOL;
BContactBit0221	:BOOL;
BContactBit0222	:BOOL;
BContactBit0223	:BOOL;
BContactBit0224	:BOOL;
BContactBit0225	:BOOL;
BContactBit0226	:BOOL;
BContactBit0227	:BOOL;
BContactBit0228	:BOOL;
BContactBit0229	:BOOL;
BContactBit0230	:BOOL;
BContactBit0231	:BOOL;
BContactBit0232	:BOOL;
BContactBit0233	:BOOL;
BContactBit0234	:BOOL;
BContactBit0235	:BOOL;
BContactBit0236	:BOOL;
BContactBit0237	:BOOL;
BContactBit0238	:BOOL;
BContactBit0239	:BOOL;
BContactBit0240	:BOOL;
BContactBit0241	:BOOL;
BContactBit0242	:BOOL;
BContactBit0243	:BOOL;
BContactBit0244	:BOOL;
BContactBit0245	:BOOL;
BContactBit0246	:BOOL;
BContactBit0247	:BOOL;
BContactBit0248	:BOOL;
BContactBit0249	:BOOL;
BContactBit0250	:BOOL;
BContactBit0251	:BOOL;
BContactBit0252	:BOOL;
BContactBit0253	:BOOL;
BContactBit0254	:BOOL;
BContactBit0255	:BOOL;
BContactBit0256	:BOOL;
BContactBit0257	:BOOL;
BContactBit0258	:BOOL;
BContactBit0259	:BOOL;
BContactBit0260	:BOOL;
BContactBit0261	:BOOL;
BContactBit0262	:BOOL;
BContactBit0263	:BOOL;
BContactBit0264	:BOOL;
BContactBit0265	:BOOL;
BContactBit0266	:BOOL;
BContactBit0267	:BOOL;
BContactBit0268	:BOOL;
BContactBit0269	:BOOL;
BContactBit0270	:BOOL;
BContactBit0271	:BOOL;
BContactBit0272	:BOOL;
BContactBit0273	:BOOL;
BContactBit0274	:BOOL;
BContactBit0275	:BOOL;
BContactBit0276	:BOOL;
BContactBit0277	:BOOL;
BContactBit0278	:BOOL;
BContactBit0279	:BOOL;
BContactBit0280	:BOOL;
BContactBit0281	:BOOL;
BContactBit0282	:BOOL;
BContactBit0283	:BOOL;
BContactBit0284	:BOOL;
BContactBit0285	:BOOL;
BContactBit0286	:BOOL;
BContactBit0287	:BOOL;
BContactBit0288	:BOOL;
BContactBit0289	:BOOL;
BContactBit0290	:BOOL;
BContactBit0291	:BOOL;
BContactBit0292	:BOOL;
BContactBit0293	:BOOL;
BContactBit0294	:BOOL;
BContactBit0295	:BOOL;
BContactBit0296	:BOOL;
BContactBit0297	:BOOL;
BContactBit0298	:BOOL;
BContactBit0299	:BOOL;
BContactBit0300	:BOOL;
BContactBit0301	:BOOL;
BContactBit0302	:BOOL;
BContactBit0303	:BOOL;
BContactBit0304	:BOOL;
BContactBit0305	:BOOL;
BContactBit0306	:BOOL;
BContactBit0307	:BOOL;
BContactBit0308	:BOOL;
BContactBit0309	:BOOL;
BContactBit0310	:BOOL;
BContactBit0311	:BOOL;
BContactBit0312	:BOOL;
BContactBit0313	:BOOL;
BContactBit0314	:BOOL;
BContactBit0315	:BOOL;
BContactBit0316	:BOOL;
BContactBit0317	:BOOL;
BContactBit0318	:BOOL;
BContactBit0319	:BOOL;
BContactBit0320	:BOOL;
BContactBit0321	:BOOL;
BContactBit0322	:BOOL;
BContactBit0323	:BOOL;
BContactBit0324	:BOOL;
BContactBit0325	:BOOL;
BContactBit0326	:BOOL;
BContactBit0327	:BOOL;
BContactBit0328	:BOOL;
BContactBit0329	:BOOL;
BContactBit0330	:BOOL;
BContactBit0331	:BOOL;
BContactBit0332	:BOOL;
BContactBit0333	:BOOL;
BContactBit0334	:BOOL;
BContactBit0335	:BOOL;
BContactBit0336	:BOOL;
BContactBit0337	:BOOL;
BContactBit0338	:BOOL;
BContactBit0339	:BOOL;
BContactBit0340	:BOOL;
BContactBit0341	:BOOL;
BContactBit0342	:BOOL;
BContactBit0343	:BOOL;
BContactBit0344	:BOOL;
BContactBit0345	:BOOL;
BContactBit0346	:BOOL;
BContactBit0347	:BOOL;
BContactBit0348	:BOOL;
BContactBit0349	:BOOL;
BContactBit0350	:BOOL;
BContactBit0351	:BOOL;
BContactBit0352	:BOOL;
BContactBit0353	:BOOL;
BContactBit0354	:BOOL;
BContactBit0355	:BOOL;
BContactBit0356	:BOOL;
BContactBit0357	:BOOL;
BContactBit0358	:BOOL;
BContactBit0359	:BOOL;
BContactBit0360	:BOOL;
BContactBit0361	:BOOL;
BContactBit0362	:BOOL;
BContactBit0363	:BOOL;
BContactBit0364	:BOOL;
BContactBit0365	:BOOL;
BContactBit0366	:BOOL;
BContactBit0367	:BOOL;
BContactBit0368	:BOOL;
BContactBit0369	:BOOL;
BContactBit0370	:BOOL;
BContactBit0371	:BOOL;
BContactBit0372	:BOOL;
BContactBit0373	:BOOL;
BContactBit0374	:BOOL;
BContactBit0375	:BOOL;
BContactBit0376	:BOOL;
BContactBit0377	:BOOL;
BContactBit0378	:BOOL;
BContactBit0379	:BOOL;
BContactBit0380	:BOOL;
BContactBit0381	:BOOL;
BContactBit0382	:BOOL;
BContactBit0383	:BOOL;
BContactBit0384	:BOOL;
BContactBit0385	:BOOL;
BContactBit0386	:BOOL;
BContactBit0387	:BOOL;
BContactBit0388	:BOOL;
BContactBit0389	:BOOL;
BContactBit0390	:BOOL;
BContactBit0391	:BOOL;
BContactBit0392	:BOOL;
BContactBit0393	:BOOL;
BContactBit0394	:BOOL;
BContactBit0395	:BOOL;
BContactBit0396	:BOOL;
BContactBit0397	:BOOL;
BContactBit0398	:BOOL;
BContactBit0399	:BOOL;
BContactBit0400	:BOOL;
BContactBit0401	:BOOL;
BContactBit0402	:BOOL;
BContactBit0403	:BOOL;
BContactBit0404	:BOOL;
BContactBit0405	:BOOL;
BContactBit0406	:BOOL;
BContactBit0407	:BOOL;
BContactBit0408	:BOOL;
BContactBit0409	:BOOL;
BContactBit0410	:BOOL;
BContactBit0411	:BOOL;
BContactBit0412	:BOOL;
BContactBit0413	:BOOL;
BContactBit0414	:BOOL;
BContactBit0415	:BOOL;
BContactBit0416	:BOOL;
BContactBit0417	:BOOL;
BContactBit0418	:BOOL;
BContactBit0419	:BOOL;
BContactBit0420	:BOOL;
BContactBit0421	:BOOL;
BContactBit0422	:BOOL;
BContactBit0423	:BOOL;
BContactBit0424	:BOOL;
BContactBit0425	:BOOL;
BContactBit0426	:BOOL;
BContactBit0427	:BOOL;
BContactBit0428	:BOOL;
BContactBit0429	:BOOL;
BContactBit0430	:BOOL;
BContactBit0431	:BOOL;
BContactBit0432	:BOOL;
BContactBit0433	:BOOL;
BContactBit0434	:BOOL;
BContactBit0435	:BOOL;
BContactBit0436	:BOOL;
BContactBit0437	:BOOL;
BContactBit0438	:BOOL;
BContactBit0439	:BOOL;
BContactBit0440	:BOOL;
BContactBit0441	:BOOL;
BContactBit0442	:BOOL;
BContactBit0443	:BOOL;
BContactBit0444	:BOOL;
BContactBit0445	:BOOL;
BContactBit0446	:BOOL;
BContactBit0447	:BOOL;
BContactBit0448	:BOOL;
BContactBit0449	:BOOL;
BContactBit0450	:BOOL;
BContactBit0451	:BOOL;
BContactBit0452	:BOOL;
BContactBit0453	:BOOL;
BContactBit0454	:BOOL;
BContactBit0455	:BOOL;
BContactBit0456	:BOOL;
BContactBit0457	:BOOL;
BContactBit0458	:BOOL;
BContactBit0459	:BOOL;
BContactBit0460	:BOOL;
BContactBit0461	:BOOL;
BContactBit0462	:BOOL;
BContactBit0463	:BOOL;
BContactBit0464	:BOOL;
BContactBit0465	:BOOL;
BContactBit0466	:BOOL;
BContactBit0467	:BOOL;
BContactBit0468	:BOOL;
BContactBit0469	:BOOL;
BContactBit0470	:BOOL;
BContactBit0471	:BOOL;
BContactBit0472	:BOOL;
BContactBit0473	:BOOL;
BContactBit0474	:BOOL;
BContactBit0475	:BOOL;
BContactBit0476	:BOOL;
BContactBit0477	:BOOL;
BContactBit0478	:BOOL;
BContactBit0479	:BOOL;
BContactBit0480	:BOOL;
BContactBit0481	:BOOL;
BContactBit0482	:BOOL;
BContactBit0483	:BOOL;
BContactBit0484	:BOOL;
BContactBit0485	:BOOL;
BContactBit0486	:BOOL;
BContactBit0487	:BOOL;
BContactBit0488	:BOOL;
BContactBit0489	:BOOL;
BContactBit0490	:BOOL;
BContactBit0491	:BOOL;
BContactBit0492	:BOOL;
BContactBit0493	:BOOL;
BContactBit0494	:BOOL;
BContactBit0495	:BOOL;
BContactBit0496	:BOOL;
BContactBit0497	:BOOL;
BContactBit0498	:BOOL;
BContactBit0499	:BOOL;
BContactBit0500	:BOOL;

CoilBit0000	:BOOL;
CoilBit0001	:BOOL;
CoilBit0002	:BOOL;
CoilBit0003	:BOOL;
CoilBit0004	:BOOL;
CoilBit0005	:BOOL;
CoilBit0006	:BOOL;
CoilBit0007	:BOOL;
CoilBit0008	:BOOL;
CoilBit0009	:BOOL;
CoilBit0010	:BOOL;
CoilBit0011	:BOOL;
CoilBit0012	:BOOL;
CoilBit0013	:BOOL;
CoilBit0014	:BOOL;
CoilBit0015	:BOOL;
CoilBit0016	:BOOL;
CoilBit0017	:BOOL;
CoilBit0018	:BOOL;
CoilBit0019	:BOOL;
CoilBit0020	:BOOL;
CoilBit0021	:BOOL;
CoilBit0022	:BOOL;
CoilBit0023	:BOOL;
CoilBit0024	:BOOL;
CoilBit0025	:BOOL;
CoilBit0026	:BOOL;
CoilBit0027	:BOOL;
CoilBit0028	:BOOL;
CoilBit0029	:BOOL;
CoilBit0030	:BOOL;
CoilBit0031	:BOOL;
CoilBit0032	:BOOL;
CoilBit0033	:BOOL;
CoilBit0034	:BOOL;
CoilBit0035	:BOOL;
CoilBit0036	:BOOL;
CoilBit0037	:BOOL;
CoilBit0038	:BOOL;
CoilBit0039	:BOOL;
CoilBit0040	:BOOL;
CoilBit0041	:BOOL;
CoilBit0042	:BOOL;
CoilBit0043	:BOOL;
CoilBit0044	:BOOL;
CoilBit0045	:BOOL;
CoilBit0046	:BOOL;
CoilBit0047	:BOOL;
CoilBit0048	:BOOL;
CoilBit0049	:BOOL;
CoilBit0050	:BOOL;
CoilBit0051	:BOOL;
CoilBit0052	:BOOL;
CoilBit0053	:BOOL;
CoilBit0054	:BOOL;
CoilBit0055	:BOOL;
CoilBit0056	:BOOL;
CoilBit0057	:BOOL;
CoilBit0058	:BOOL;
CoilBit0059	:BOOL;
CoilBit0060	:BOOL;
CoilBit0061	:BOOL;
CoilBit0062	:BOOL;
CoilBit0063	:BOOL;
CoilBit0064	:BOOL;
CoilBit0065	:BOOL;
CoilBit0066	:BOOL;
CoilBit0067	:BOOL;
CoilBit0068	:BOOL;
CoilBit0069	:BOOL;
CoilBit0070	:BOOL;
CoilBit0071	:BOOL;
CoilBit0072	:BOOL;
CoilBit0073	:BOOL;
CoilBit0074	:BOOL;
CoilBit0075	:BOOL;
CoilBit0076	:BOOL;
CoilBit0077	:BOOL;
CoilBit0078	:BOOL;
CoilBit0079	:BOOL;
CoilBit0080	:BOOL;
CoilBit0081	:BOOL;
CoilBit0082	:BOOL;
CoilBit0083	:BOOL;
CoilBit0084	:BOOL;
CoilBit0085	:BOOL;
CoilBit0086	:BOOL;
CoilBit0087	:BOOL;
CoilBit0088	:BOOL;
CoilBit0089	:BOOL;
CoilBit0090	:BOOL;
CoilBit0091	:BOOL;
CoilBit0092	:BOOL;
CoilBit0093	:BOOL;
CoilBit0094	:BOOL;
CoilBit0095	:BOOL;
CoilBit0096	:BOOL;
CoilBit0097	:BOOL;
CoilBit0098	:BOOL;
CoilBit0099	:BOOL;
CoilBit0100	:BOOL;

END_VAR

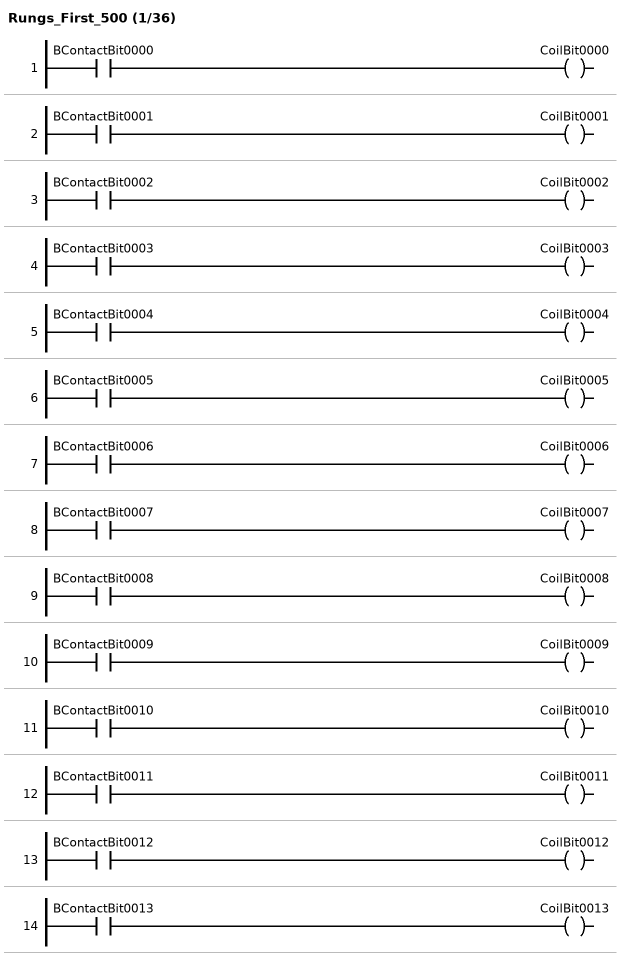
// NETWORK 1
CoilBit0000 := BContactBit0000;

// NETWORK 2
CoilBit0001 := BContactBit0001;

// NETWORK 3
CoilBit0002 := BContactBit0002;

// NETWORK 4
CoilBit0003 := BContactBit0003;

// NETWORK 5
CoilBit0004 := BContactBit0004;

// NETWORK 6
CoilBit0005 := BContactBit0005;

// NETWORK 7
CoilBit0006 := BContactBit0006;

// NETWORK 8
CoilBit0007 := BContactBit0007;

// NETWORK 9
CoilBit0008 := BContactBit0008;

// NETWORK 10
CoilBit0009 := BContactBit0009;

// NETWORK 11
CoilBit0010 := BContactBit0010;

// NETWORK 12
CoilBit0011 := BContactBit0011;

// NETWORK 13
CoilBit0012 := BContactBit0012;

// NETWORK 14
CoilBit0013 := BContactBit0013;

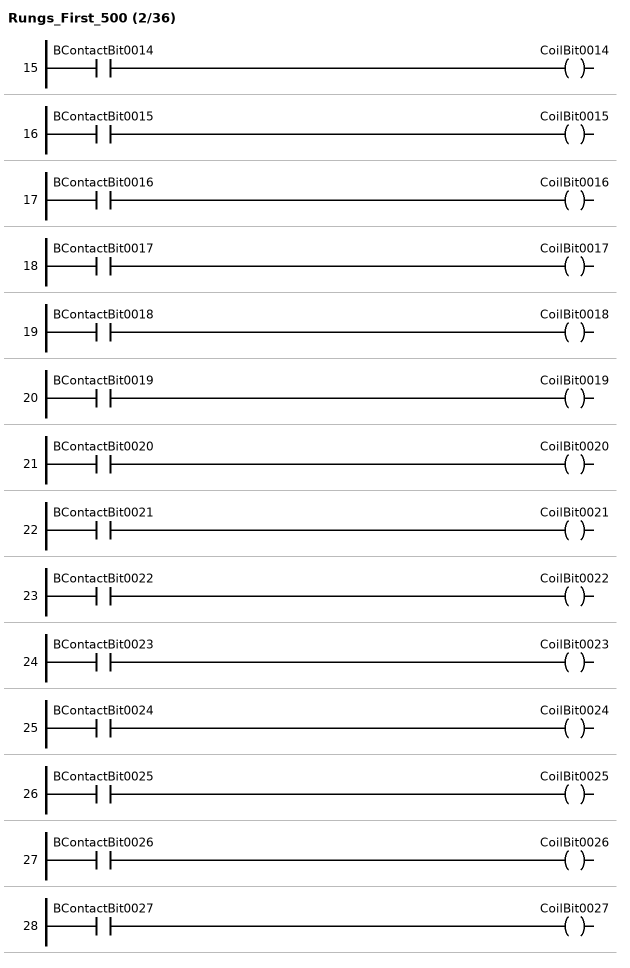
// NETWORK 15
CoilBit0014 := BContactBit0014;

// NETWORK 16
CoilBit0015 := BContactBit0015;

// NETWORK 17
CoilBit0016 := BContactBit0016;

// NETWORK 18
CoilBit0017 := BContactBit0017;

// NETWORK 19
CoilBit0018 := BContactBit0018;

// NETWORK 20
CoilBit0019 := BContactBit0019;

// NETWORK 21
CoilBit0020 := BContactBit0020;

// NETWORK 22
CoilBit0021 := BContactBit0021;

// NETWORK 23
CoilBit0022 := BContactBit0022;

// NETWORK 24
CoilBit0023 := BContactBit0023;

// NETWORK 25
CoilBit0024 := BContactBit0024;

// NETWORK 26
CoilBit0025 := BContactBit0025;

// NETWORK 27
CoilBit0026 := BContactBit0026;

// NETWORK 28
CoilBit0027 := BContactBit0027;

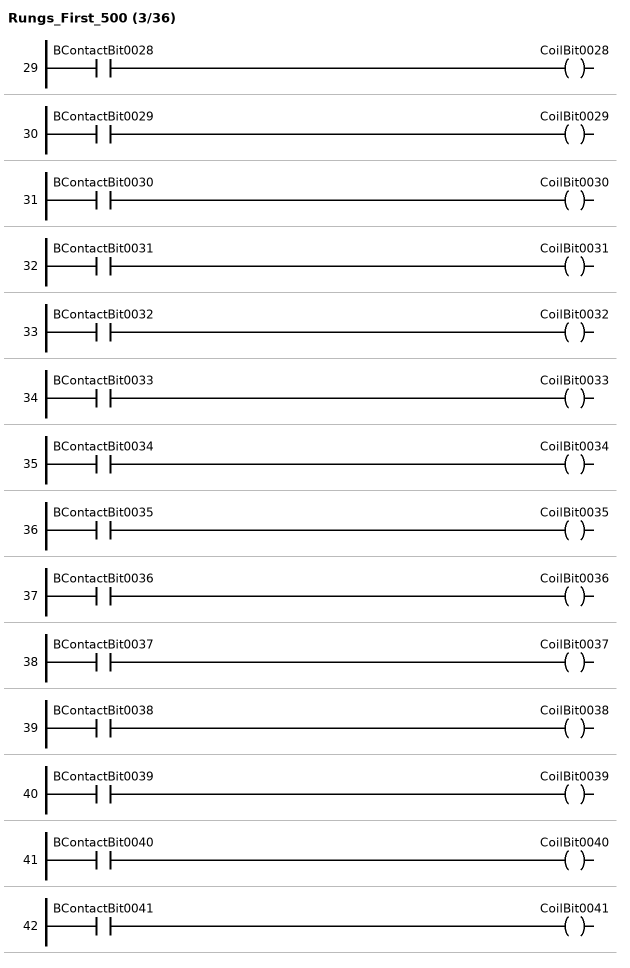
// NETWORK 29
CoilBit0028 := BContactBit0028;

// NETWORK 30
CoilBit0029 := BContactBit0029;

// NETWORK 31
CoilBit0030 := BContactBit0030;

// NETWORK 32
CoilBit0031 := BContactBit0031;

// NETWORK 33
CoilBit0032 := BContactBit0032;

// NETWORK 34
CoilBit0033 := BContactBit0033;

// NETWORK 35
CoilBit0034 := BContactBit0034;

// NETWORK 36
CoilBit0035 := BContactBit0035;

// NETWORK 37
CoilBit0036 := BContactBit0036;

// NETWORK 38
CoilBit0037 := BContactBit0037;

// NETWORK 39
CoilBit0038 := BContactBit0038;

// NETWORK 40
CoilBit0039 := BContactBit0039;

// NETWORK 41
CoilBit0040 := BContactBit0040;

// NETWORK 42
CoilBit0041 := BContactBit0041;

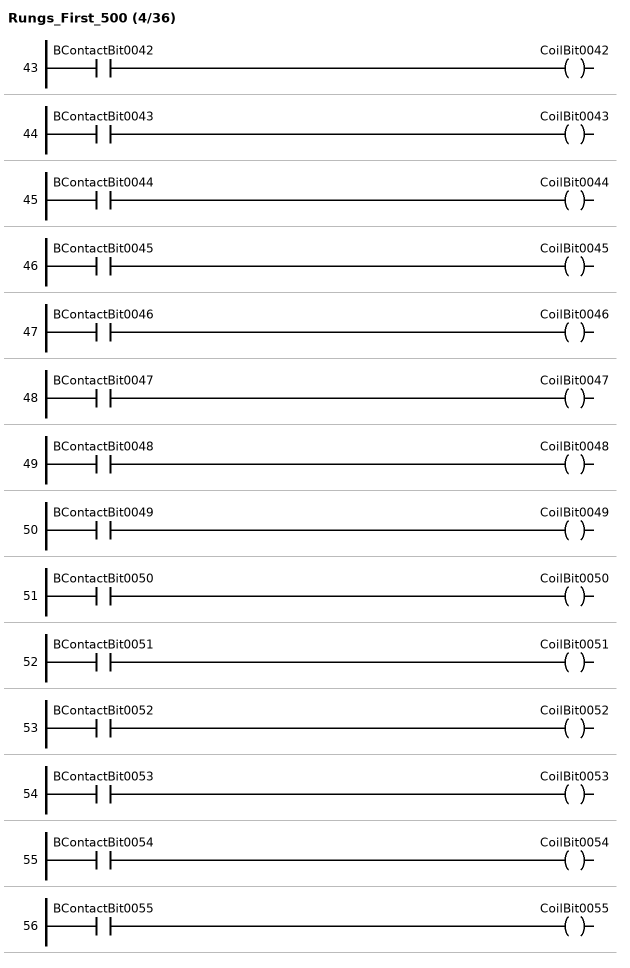
// NETWORK 43
CoilBit0042 := BContactBit0042;

// NETWORK 44
CoilBit0043 := BContactBit0043;

// NETWORK 45
CoilBit0044 := BContactBit0044;

// NETWORK 46
CoilBit0045 := BContactBit0045;

// NETWORK 47
CoilBit0046 := BContactBit0046;

// NETWORK 48
CoilBit0047 := BContactBit0047;

// NETWORK 49
CoilBit0048 := BContactBit0048;

// NETWORK 50
CoilBit0049 := BContactBit0049;

// NETWORK 51
CoilBit0050 := BContactBit0050;

// NETWORK 52
CoilBit0051 := BContactBit0051;

// NETWORK 53
CoilBit0052 := BContactBit0052;

// NETWORK 54
CoilBit0053 := BContactBit0053;

// NETWORK 55
CoilBit0054 := BContactBit0054;

// NETWORK 56
CoilBit0055 := BContactBit0055;

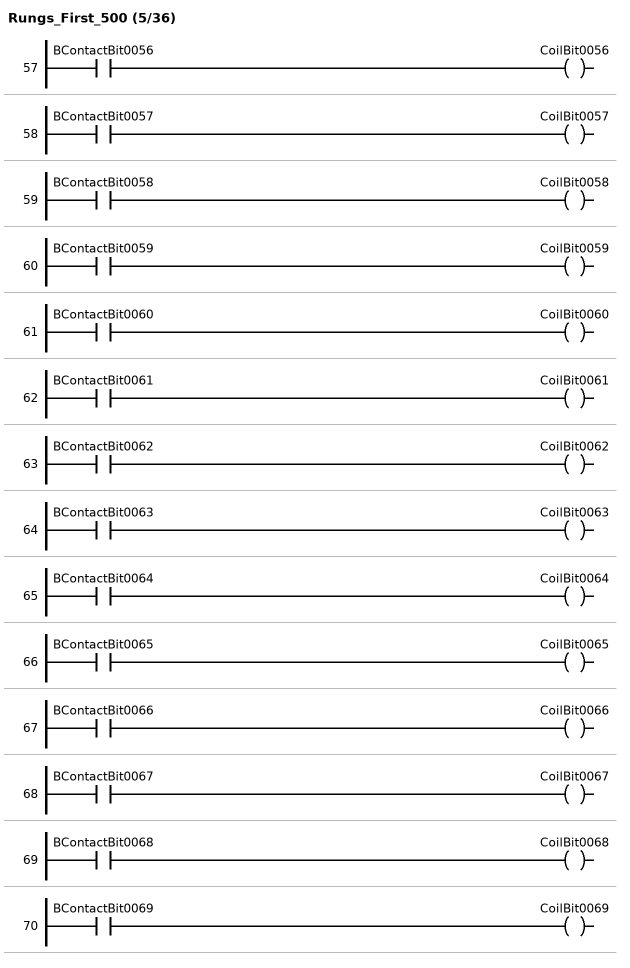
// NETWORK 57
CoilBit0056 := BContactBit0056;

// NETWORK 58
CoilBit0057 := BContactBit0057;

// NETWORK 59
CoilBit0058 := BContactBit0058;

// NETWORK 60
CoilBit0059 := BContactBit0059;

// NETWORK 61
CoilBit0060 := BContactBit0060;

// NETWORK 62
CoilBit0061 := BContactBit0061;

// NETWORK 63
CoilBit0062 := BContactBit0062;

// NETWORK 64
CoilBit0063 := BContactBit0063;

// NETWORK 65
CoilBit0064 := BContactBit0064;

// NETWORK 66
CoilBit0065 := BContactBit0065;

// NETWORK 67
CoilBit0066 := BContactBit0066;

// NETWORK 68
CoilBit0067 := BContactBit0067;

// NETWORK 69
CoilBit0068 := BContactBit0068;

// NETWORK 70
CoilBit0069 := BContactBit0069;

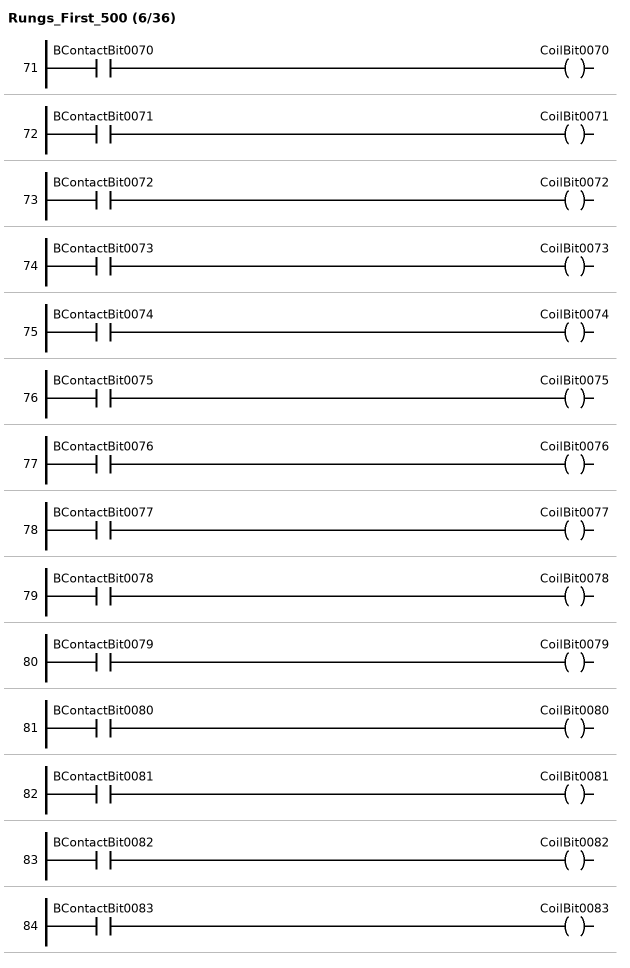
// NETWORK 71
CoilBit0070 := BContactBit0070;

// NETWORK 72
CoilBit0071 := BContactBit0071;

// NETWORK 73
CoilBit0072 := BContactBit0072;

// NETWORK 74
CoilBit0073 := BContactBit0073;

// NETWORK 75
CoilBit0074 := BContactBit0074;

// NETWORK 76
CoilBit0075 := BContactBit0075;

// NETWORK 77
CoilBit0076 := BContactBit0076;

// NETWORK 78
CoilBit0077 := BContactBit0077;

// NETWORK 79
CoilBit0078 := BContactBit0078;

// NETWORK 80
CoilBit0079 := BContactBit0079;

// NETWORK 81
CoilBit0080 := BContactBit0080;

// NETWORK 82
CoilBit0081 := BContactBit0081;

// NETWORK 83
CoilBit0082 := BContactBit0082;

// NETWORK 84
CoilBit0083 := BContactBit0083;

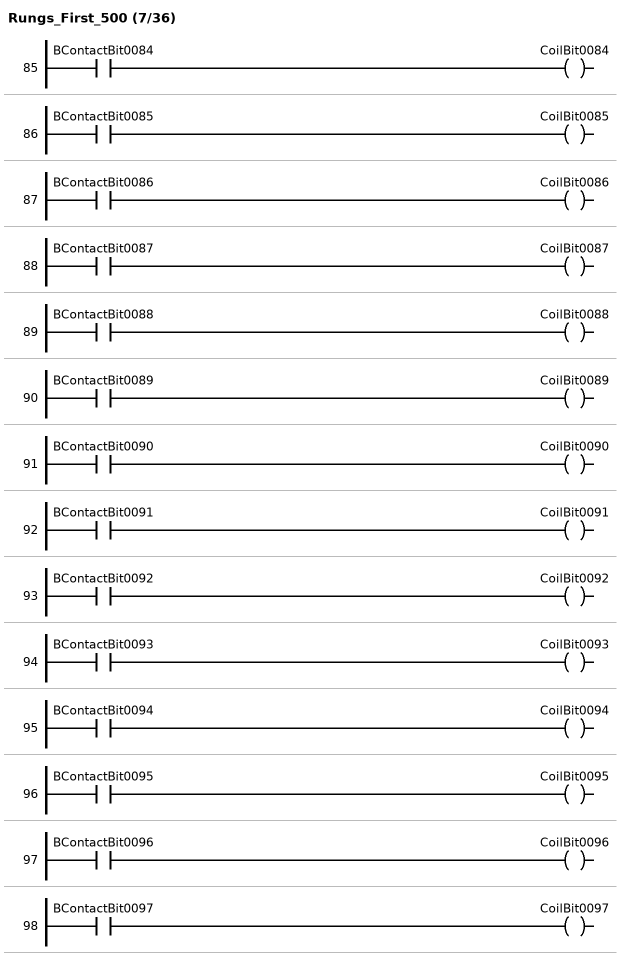
// NETWORK 85
CoilBit0084 := BContactBit0084;

// NETWORK 86
CoilBit0085 := BContactBit0085;

// NETWORK 87
CoilBit0086 := BContactBit0086;

// NETWORK 88
CoilBit0087 := BContactBit0087;

// NETWORK 89
CoilBit0088 := BContactBit0088;

// NETWORK 90
CoilBit0089 := BContactBit0089;

// NETWORK 91
CoilBit0090 := BContactBit0090;

// NETWORK 92
CoilBit0091 := BContactBit0091;

// NETWORK 93
CoilBit0092 := BContactBit0092;

// NETWORK 94
CoilBit0093 := BContactBit0093;

// NETWORK 95
CoilBit0094 := BContactBit0094;

// NETWORK 96
CoilBit0095 := BContactBit0095;

// NETWORK 97
CoilBit0096 := BContactBit0096;

// NETWORK 98
CoilBit0097 := BContactBit0097;

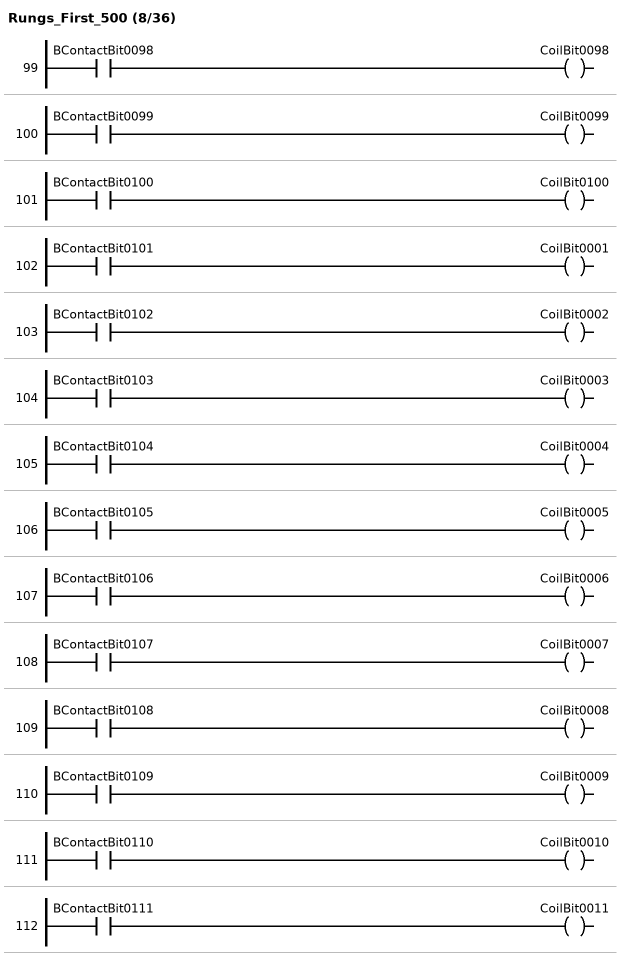
// NETWORK 99
CoilBit0098 := BContactBit0098;

// NETWORK 100
CoilBit0099 := BContactBit0099;

// NETWORK 101
CoilBit0100 := BContactBit0100;

// NETWORK 102
CoilBit0001 := BContactBit0101;

// NETWORK 103
CoilBit0002 := BContactBit0102;

// NETWORK 104
CoilBit0003 := BContactBit0103;

// NETWORK 105
CoilBit0004 := BContactBit0104;

// NETWORK 106
CoilBit0005 := BContactBit0105;

// NETWORK 107
CoilBit0006 := BContactBit0106;

// NETWORK 108
CoilBit0007 := BContactBit0107;

// NETWORK 109
CoilBit0008 := BContactBit0108;

// NETWORK 110
CoilBit0009 := BContactBit0109;

// NETWORK 111
CoilBit0010 := BContactBit0110;

// NETWORK 112
CoilBit0011 := BContactBit0111;

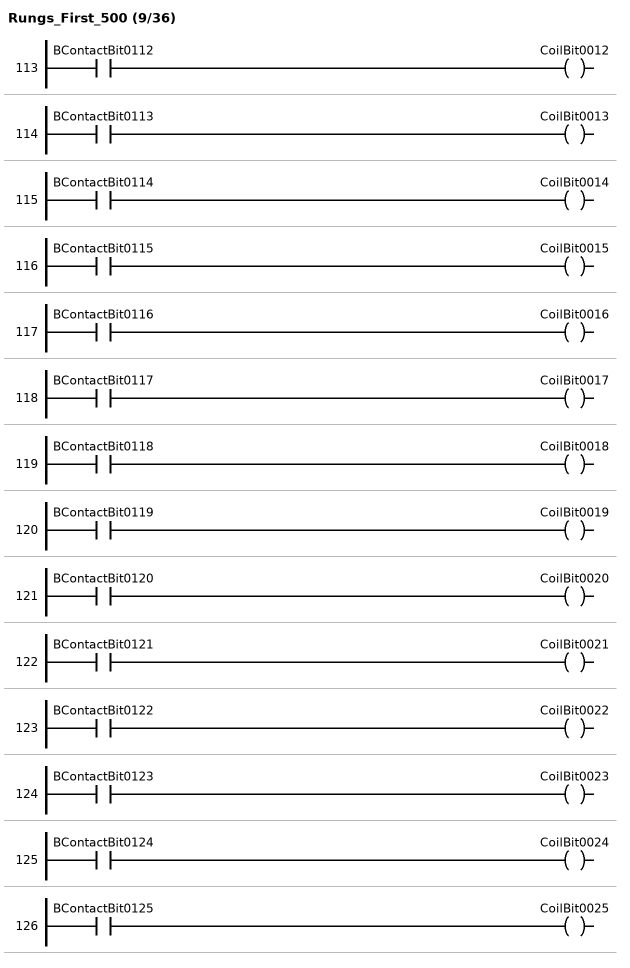
// NETWORK 113
CoilBit0012 := BContactBit0112;

// NETWORK 114
CoilBit0013 := BContactBit0113;

// NETWORK 115
CoilBit0014 := BContactBit0114;

// NETWORK 116
CoilBit0015 := BContactBit0115;

// NETWORK 117
CoilBit0016 := BContactBit0116;

// NETWORK 118
CoilBit0017 := BContactBit0117;

// NETWORK 119
CoilBit0018 := BContactBit0118;

// NETWORK 120
CoilBit0019 := BContactBit0119;

// NETWORK 121
CoilBit0020 := BContactBit0120;

// NETWORK 122
CoilBit0021 := BContactBit0121;

// NETWORK 123
CoilBit0022 := BContactBit0122;

// NETWORK 124
CoilBit0023 := BContactBit0123;

// NETWORK 125
CoilBit0024 := BContactBit0124;

// NETWORK 126
CoilBit0025 := BContactBit0125;

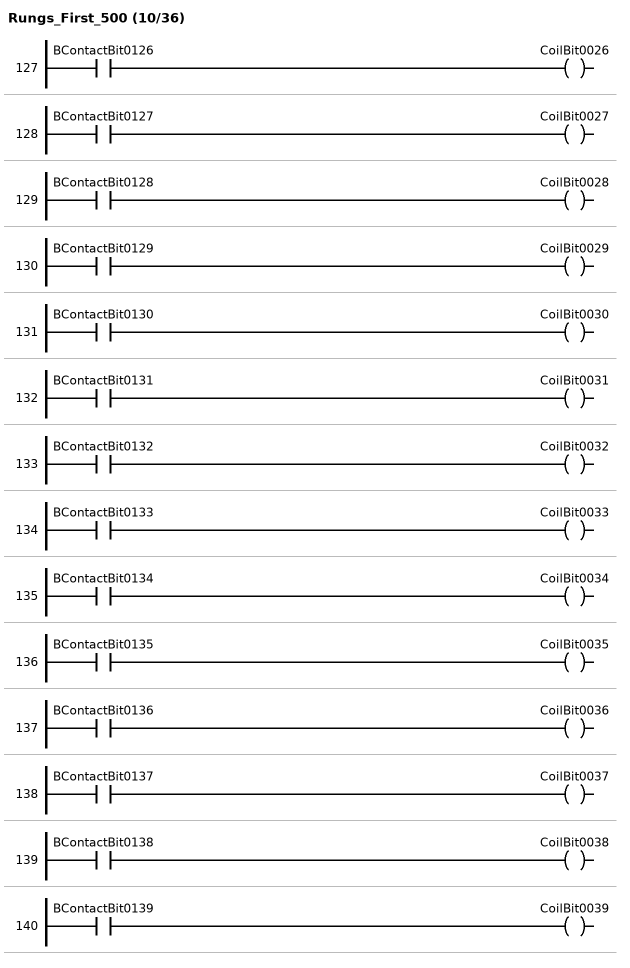
// NETWORK 127
CoilBit0026 := BContactBit0126;

// NETWORK 128
CoilBit0027 := BContactBit0127;

// NETWORK 129
CoilBit0028 := BContactBit0128;

// NETWORK 130
CoilBit0029 := BContactBit0129;

// NETWORK 131
CoilBit0030 := BContactBit0130;

// NETWORK 132
CoilBit0031 := BContactBit0131;

// NETWORK 133
CoilBit0032 := BContactBit0132;

// NETWORK 134
CoilBit0033 := BContactBit0133;

// NETWORK 135
CoilBit0034 := BContactBit0134;

// NETWORK 136
CoilBit0035 := BContactBit0135;

// NETWORK 137
CoilBit0036 := BContactBit0136;

// NETWORK 138
CoilBit0037 := BContactBit0137;

// NETWORK 139
CoilBit0038 := BContactBit0138;

// NETWORK 140
CoilBit0039 := BContactBit0139;

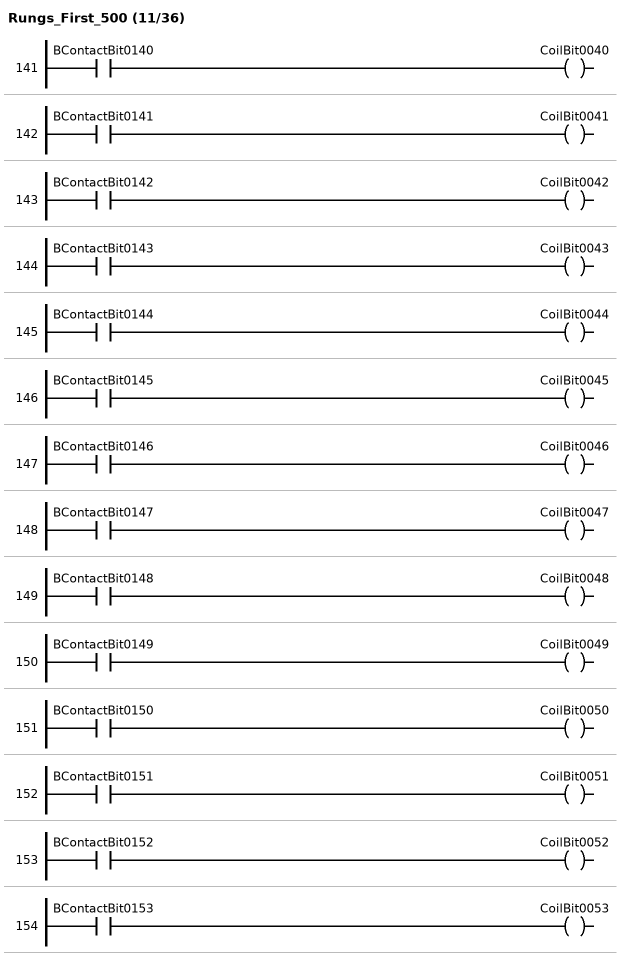
// NETWORK 141
CoilBit0040 := BContactBit0140;

// NETWORK 142
CoilBit0041 := BContactBit0141;

// NETWORK 143
CoilBit0042 := BContactBit0142;

// NETWORK 144
CoilBit0043 := BContactBit0143;

// NETWORK 145
CoilBit0044 := BContactBit0144;

// NETWORK 146
CoilBit0045 := BContactBit0145;

// NETWORK 147
CoilBit0046 := BContactBit0146;

// NETWORK 148
CoilBit0047 := BContactBit0147;

// NETWORK 149
CoilBit0048 := BContactBit0148;

// NETWORK 150
CoilBit0049 := BContactBit0149;

// NETWORK 151
CoilBit0050 := BContactBit0150;

// NETWORK 152
CoilBit0051 := BContactBit0151;

// NETWORK 153
CoilBit0052 := BContactBit0152;

// NETWORK 154
CoilBit0053 := BContactBit0153;

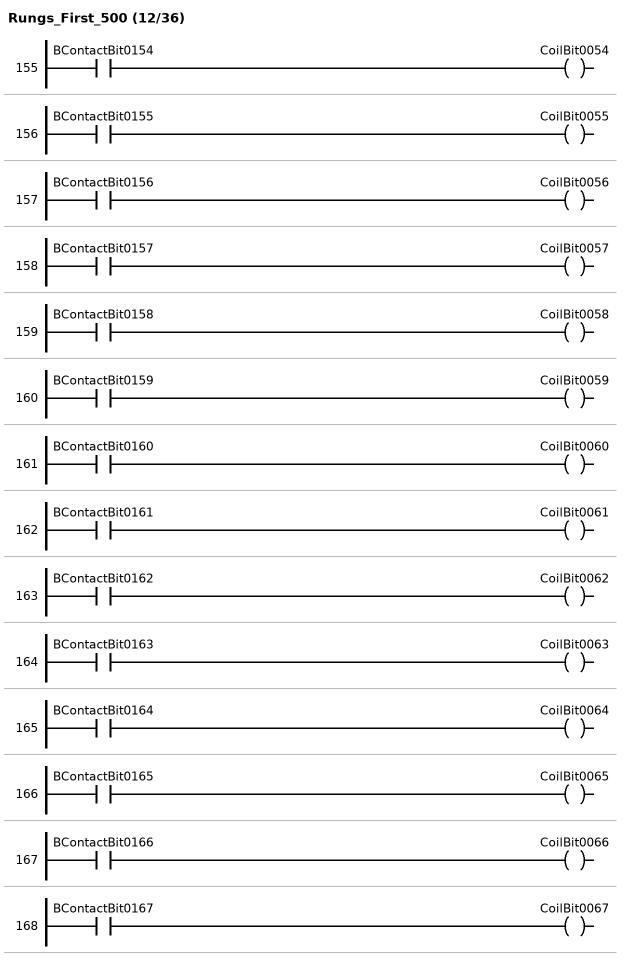
// NETWORK 155
CoilBit0054 := BContactBit0154;

// NETWORK 156
CoilBit0055 := BContactBit0155;

// NETWORK 157
CoilBit0056 := BContactBit0156;

// NETWORK 158
CoilBit0057 := BContactBit0157;

// NETWORK 159
CoilBit0058 := BContactBit0158;

// NETWORK 160
CoilBit0059 := BContactBit0159;

// NETWORK 161
CoilBit0060 := BContactBit0160;

// NETWORK 162
CoilBit0061 := BContactBit0161;

// NETWORK 163
CoilBit0062 := BContactBit0162;

// NETWORK 164
CoilBit0063 := BContactBit0163;

// NETWORK 165
CoilBit0064 := BContactBit0164;

// NETWORK 166
CoilBit0065 := BContactBit0165;

// NETWORK 167
CoilBit0066 := BContactBit0166;

// NETWORK 168
CoilBit0067 := BContactBit0167;

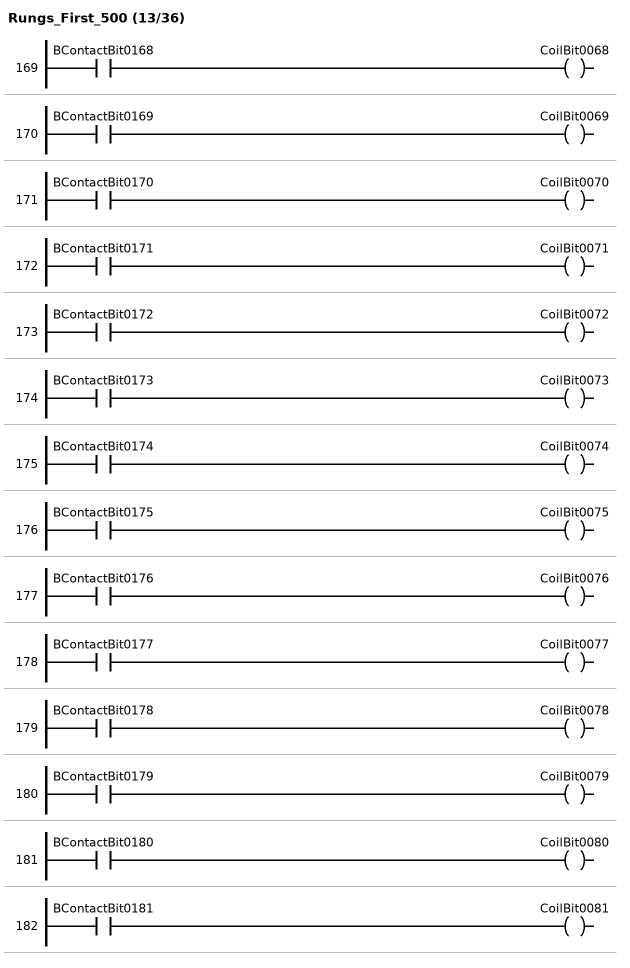
// NETWORK 169
CoilBit0068 := BContactBit0168;

// NETWORK 170
CoilBit0069 := BContactBit0169;

// NETWORK 171
CoilBit0070 := BContactBit0170;

// NETWORK 172
CoilBit0071 := BContactBit0171;

// NETWORK 173
CoilBit0072 := BContactBit0172;

// NETWORK 174
CoilBit0073 := BContactBit0173;

// NETWORK 175
CoilBit0074 := BContactBit0174;

// NETWORK 176
CoilBit0075 := BContactBit0175;

// NETWORK 177
CoilBit0076 := BContactBit0176;

// NETWORK 178
CoilBit0077 := BContactBit0177;

// NETWORK 179
CoilBit0078 := BContactBit0178;

// NETWORK 180
CoilBit0079 := BContactBit0179;

// NETWORK 181
CoilBit0080 := BContactBit0180;

// NETWORK 182
CoilBit0081 := BContactBit0181;

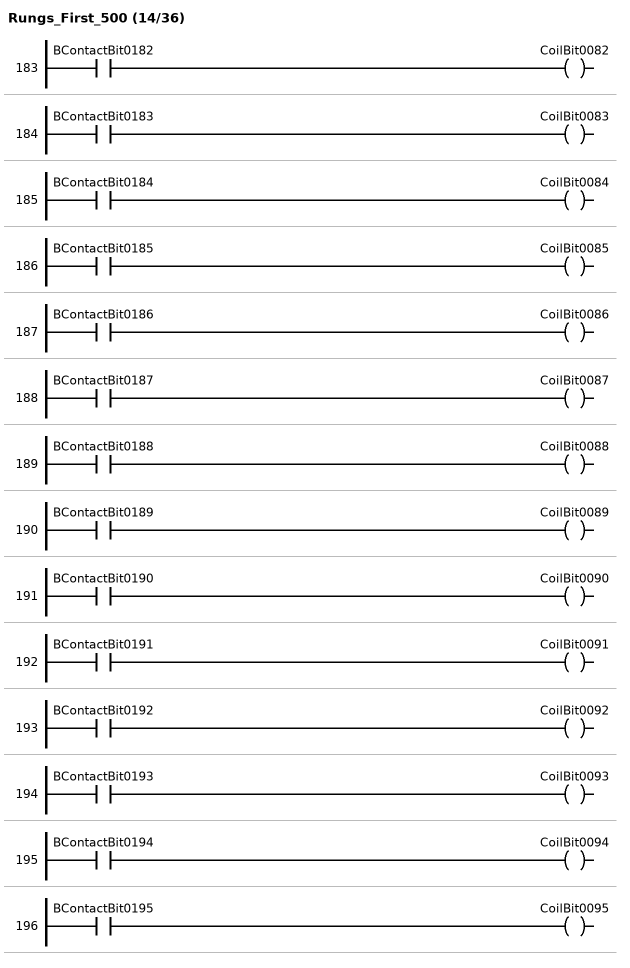
// NETWORK 183
CoilBit0082 := BContactBit0182;

// NETWORK 184
CoilBit0083 := BContactBit0183;

// NETWORK 185
CoilBit0084 := BContactBit0184;

// NETWORK 186
CoilBit0085 := BContactBit0185;

// NETWORK 187
CoilBit0086 := BContactBit0186;

// NETWORK 188
CoilBit0087 := BContactBit0187;

// NETWORK 189
CoilBit0088 := BContactBit0188;

// NETWORK 190
CoilBit0089 := BContactBit0189;

// NETWORK 191
CoilBit0090 := BContactBit0190;

// NETWORK 192
CoilBit0091 := BContactBit0191;

// NETWORK 193
CoilBit0092 := BContactBit0192;

// NETWORK 194
CoilBit0093 := BContactBit0193;

// NETWORK 195
CoilBit0094 := BContactBit0194;

// NETWORK 196
CoilBit0095 := BContactBit0195;

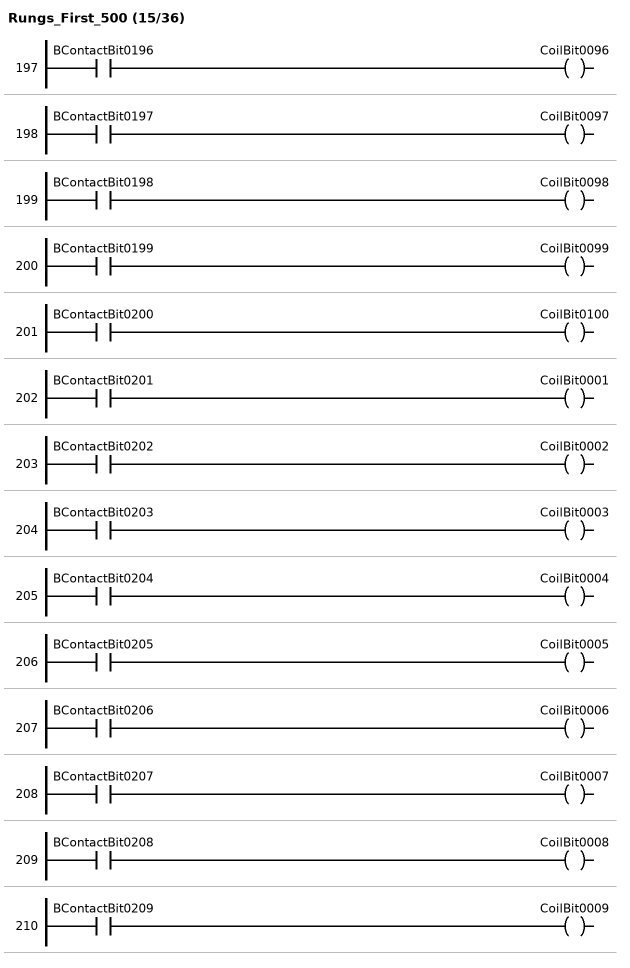
// NETWORK 197
CoilBit0096 := BContactBit0196;

// NETWORK 198
CoilBit0097 := BContactBit0197;

// NETWORK 199
CoilBit0098 := BContactBit0198;

// NETWORK 200
CoilBit0099 := BContactBit0199;

// NETWORK 201
CoilBit0100 := BContactBit0200;

// NETWORK 202
CoilBit0001 := BContactBit0201;

// NETWORK 203
CoilBit0002 := BContactBit0202;

// NETWORK 204
CoilBit0003 := BContactBit0203;

// NETWORK 205
CoilBit0004 := BContactBit0204;

// NETWORK 206
CoilBit0005 := BContactBit0205;

// NETWORK 207
CoilBit0006 := BContactBit0206;

// NETWORK 208
CoilBit0007 := BContactBit0207;

// NETWORK 209
CoilBit0008 := BContactBit0208;

// NETWORK 210
CoilBit0009 := BContactBit0209;

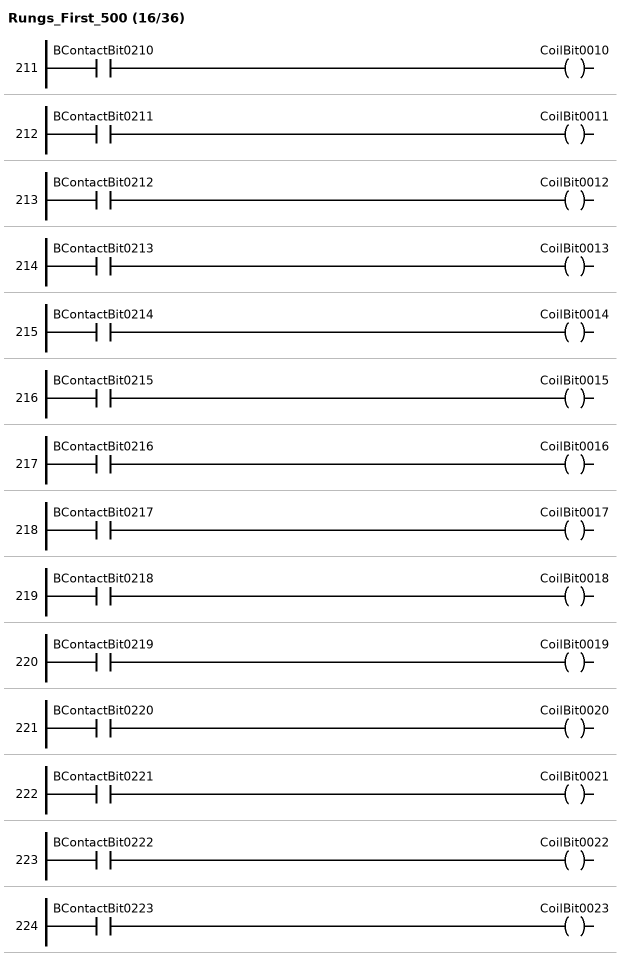
// NETWORK 211
CoilBit0010 := BContactBit0210;

// NETWORK 212
CoilBit0011 := BContactBit0211;

// NETWORK 213
CoilBit0012 := BContactBit0212;

// NETWORK 214
CoilBit0013 := BContactBit0213;

// NETWORK 215
CoilBit0014 := BContactBit0214;

// NETWORK 216
CoilBit0015 := BContactBit0215;

// NETWORK 217
CoilBit0016 := BContactBit0216;

// NETWORK 218
CoilBit0017 := BContactBit0217;

// NETWORK 219
CoilBit0018 := BContactBit0218;

// NETWORK 220
CoilBit0019 := BContactBit0219;

// NETWORK 221
CoilBit0020 := BContactBit0220;

// NETWORK 222
CoilBit0021 := BContactBit0221;

// NETWORK 223
CoilBit0022 := BContactBit0222;

// NETWORK 224
CoilBit0023 := BContactBit0223;

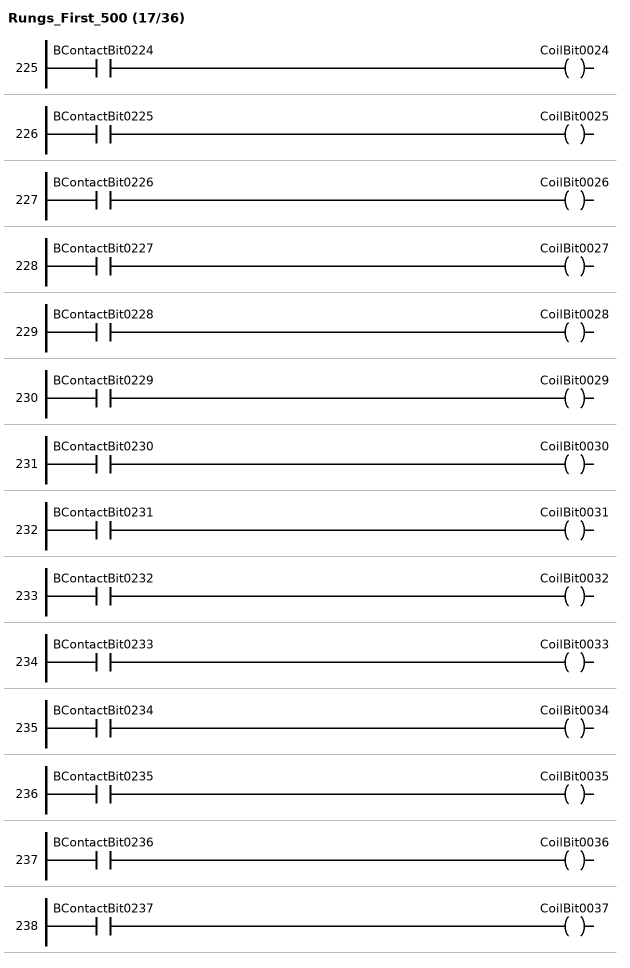
// NETWORK 225
CoilBit0024 := BContactBit0224;

// NETWORK 226
CoilBit0025 := BContactBit0225;

// NETWORK 227
CoilBit0026 := BContactBit0226;

// NETWORK 228
CoilBit0027 := BContactBit0227;

// NETWORK 229
CoilBit0028 := BContactBit0228;

// NETWORK 230
CoilBit0029 := BContactBit0229;

// NETWORK 231
CoilBit0030 := BContactBit0230;

// NETWORK 232
CoilBit0031 := BContactBit0231;

// NETWORK 233
CoilBit0032 := BContactBit0232;

// NETWORK 234
CoilBit0033 := BContactBit0233;

// NETWORK 235
CoilBit0034 := BContactBit0234;

// NETWORK 236
CoilBit0035 := BContactBit0235;

// NETWORK 237
CoilBit0036 := BContactBit0236;

// NETWORK 238
CoilBit0037 := BContactBit0237;

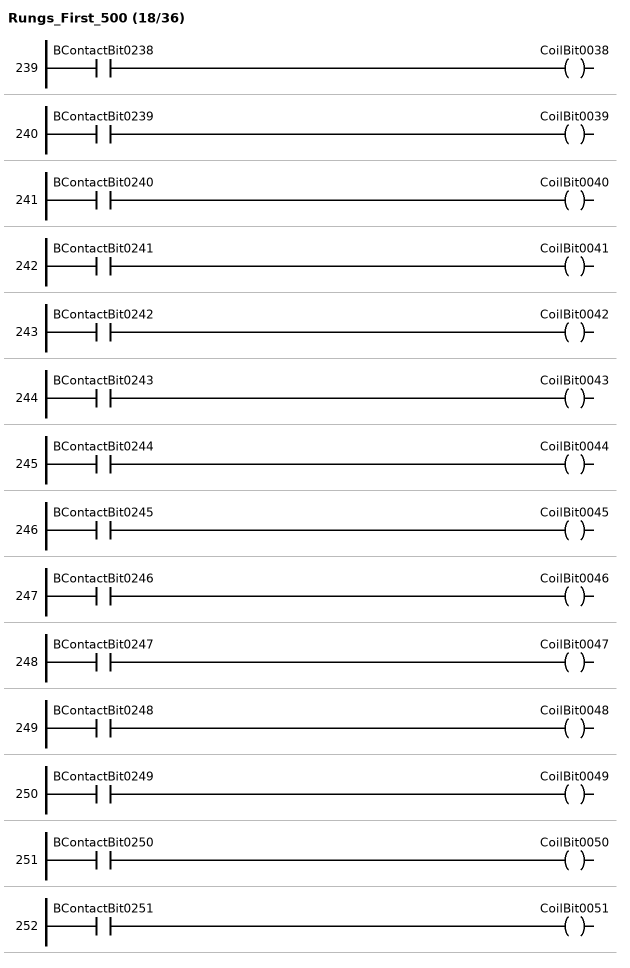
// NETWORK 239
CoilBit0038 := BContactBit0238;

// NETWORK 240
CoilBit0039 := BContactBit0239;

// NETWORK 241
CoilBit0040 := BContactBit0240;

// NETWORK 242
CoilBit0041 := BContactBit0241;

// NETWORK 243
CoilBit0042 := BContactBit0242;

// NETWORK 244
CoilBit0043 := BContactBit0243;

// NETWORK 245
CoilBit0044 := BContactBit0244;

// NETWORK 246
CoilBit0045 := BContactBit0245;

// NETWORK 247
CoilBit0046 := BContactBit0246;

// NETWORK 248
CoilBit0047 := BContactBit0247;

// NETWORK 249
CoilBit0048 := BContactBit0248;

// NETWORK 250
CoilBit0049 := BContactBit0249;

// NETWORK 251
CoilBit0050 := BContactBit0250;

// NETWORK 252
CoilBit0051 := BContactBit0251;

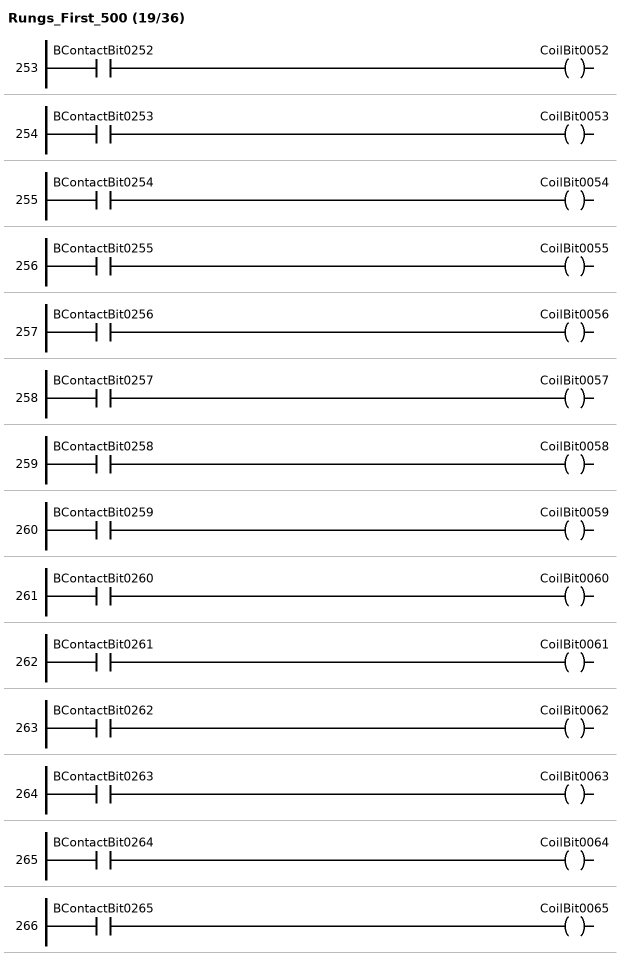
// NETWORK 253
CoilBit0052 := BContactBit0252;

// NETWORK 254
CoilBit0053 := BContactBit0253;

// NETWORK 255
CoilBit0054 := BContactBit0254;

// NETWORK 256
CoilBit0055 := BContactBit0255;

// NETWORK 257
CoilBit0056 := BContactBit0256;

// NETWORK 258
CoilBit0057 := BContactBit0257;

// NETWORK 259
CoilBit0058 := BContactBit0258;

// NETWORK 260
CoilBit0059 := BContactBit0259;

// NETWORK 261
CoilBit0060 := BContactBit0260;

// NETWORK 262
CoilBit0061 := BContactBit0261;

// NETWORK 263
CoilBit0062 := BContactBit0262;

// NETWORK 264
CoilBit0063 := BContactBit0263;

// NETWORK 265
CoilBit0064 := BContactBit0264;

// NETWORK 266
CoilBit0065 := BContactBit0265;

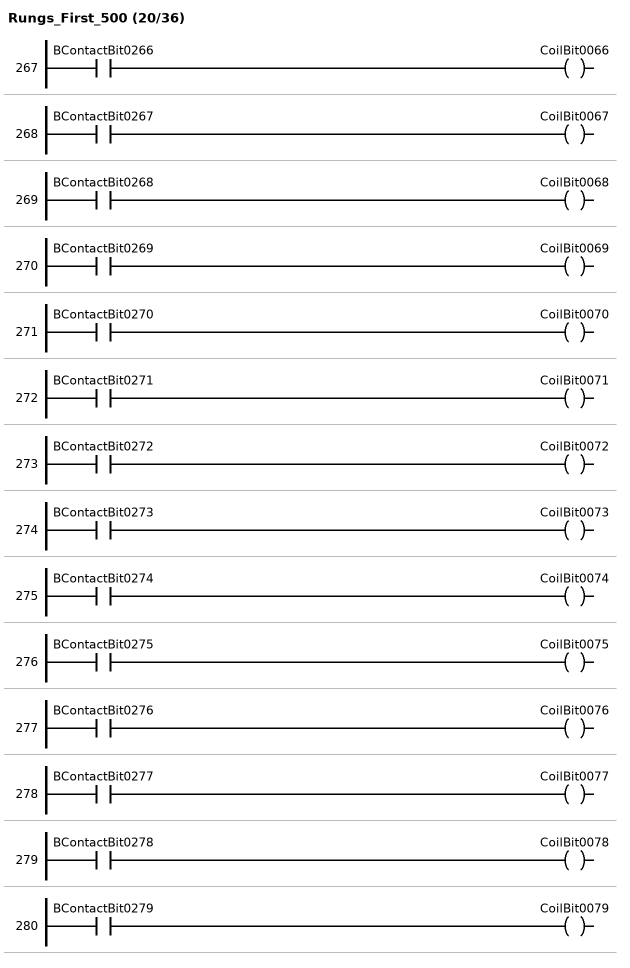
// NETWORK 267
CoilBit0066 := BContactBit0266;

// NETWORK 268
CoilBit0067 := BContactBit0267;

// NETWORK 269
CoilBit0068 := BContactBit0268;

// NETWORK 270
CoilBit0069 := BContactBit0269;

// NETWORK 271
CoilBit0070 := BContactBit0270;

// NETWORK 272
CoilBit0071 := BContactBit0271;

// NETWORK 273
CoilBit0072 := BContactBit0272;

// NETWORK 274
CoilBit0073 := BContactBit0273;

// NETWORK 275
CoilBit0074 := BContactBit0274;

// NETWORK 276
CoilBit0075 := BContactBit0275;

// NETWORK 277
CoilBit0076 := BContactBit0276;

// NETWORK 278
CoilBit0077 := BContactBit0277;

// NETWORK 279
CoilBit0078 := BContactBit0278;

// NETWORK 280
CoilBit0079 := BContactBit0279;

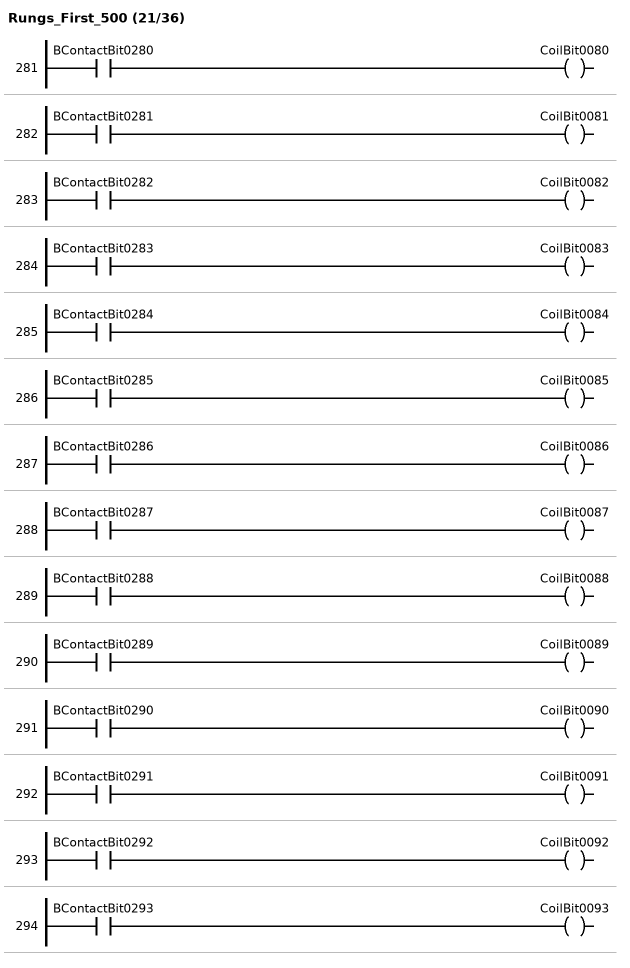
// NETWORK 281
CoilBit0080 := BContactBit0280;

// NETWORK 282
CoilBit0081 := BContactBit0281;

// NETWORK 283
CoilBit0082 := BContactBit0282;

// NETWORK 284
CoilBit0083 := BContactBit0283;

// NETWORK 285
CoilBit0084 := BContactBit0284;

// NETWORK 286
CoilBit0085 := BContactBit0285;

// NETWORK 287
CoilBit0086 := BContactBit0286;

// NETWORK 288
CoilBit0087 := BContactBit0287;

// NETWORK 289
CoilBit0088 := BContactBit0288;

// NETWORK 290
CoilBit0089 := BContactBit0289;

// NETWORK 291
CoilBit0090 := BContactBit0290;

// NETWORK 292
CoilBit0091 := BContactBit0291;

// NETWORK 293
CoilBit0092 := BContactBit0292;

// NETWORK 294
CoilBit0093 := BContactBit0293;

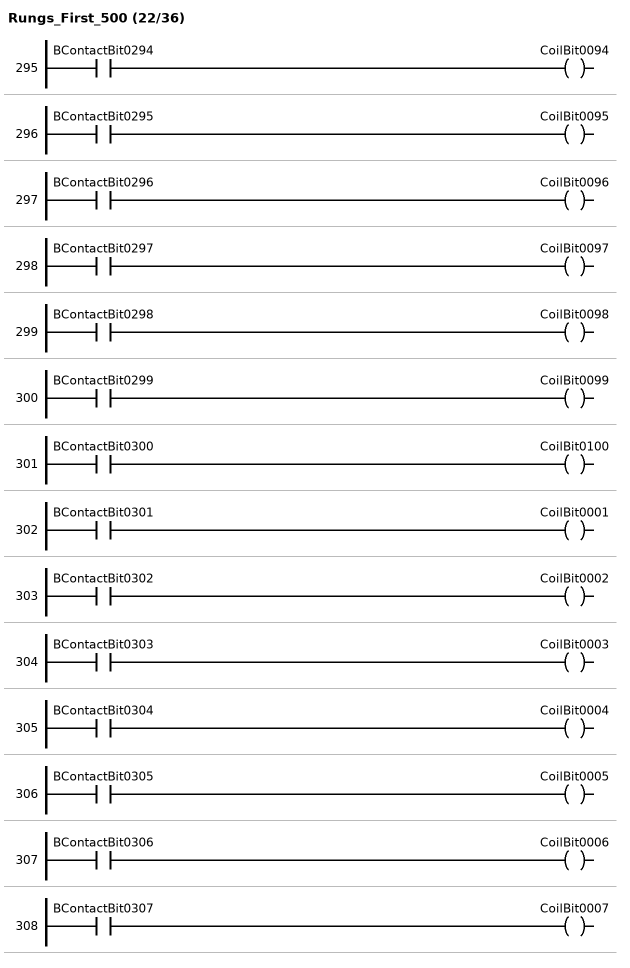
// NETWORK 295
CoilBit0094 := BContactBit0294;

// NETWORK 296
CoilBit0095 := BContactBit0295;

// NETWORK 297
CoilBit0096 := BContactBit0296;

// NETWORK 298
CoilBit0097 := BContactBit0297;

// NETWORK 299
CoilBit0098 := BContactBit0298;

// NETWORK 300
CoilBit0099 := BContactBit0299;

// NETWORK 301
CoilBit0100 := BContactBit0300;

// NETWORK 302
CoilBit0001 := BContactBit0301;

// NETWORK 303
CoilBit0002 := BContactBit0302;

// NETWORK 304
CoilBit0003 := BContactBit0303;

// NETWORK 305
CoilBit0004 := BContactBit0304;

// NETWORK 306
CoilBit0005 := BContactBit0305;

// NETWORK 307
CoilBit0006 := BContactBit0306;

// NETWORK 308
CoilBit0007 := BContactBit0307;

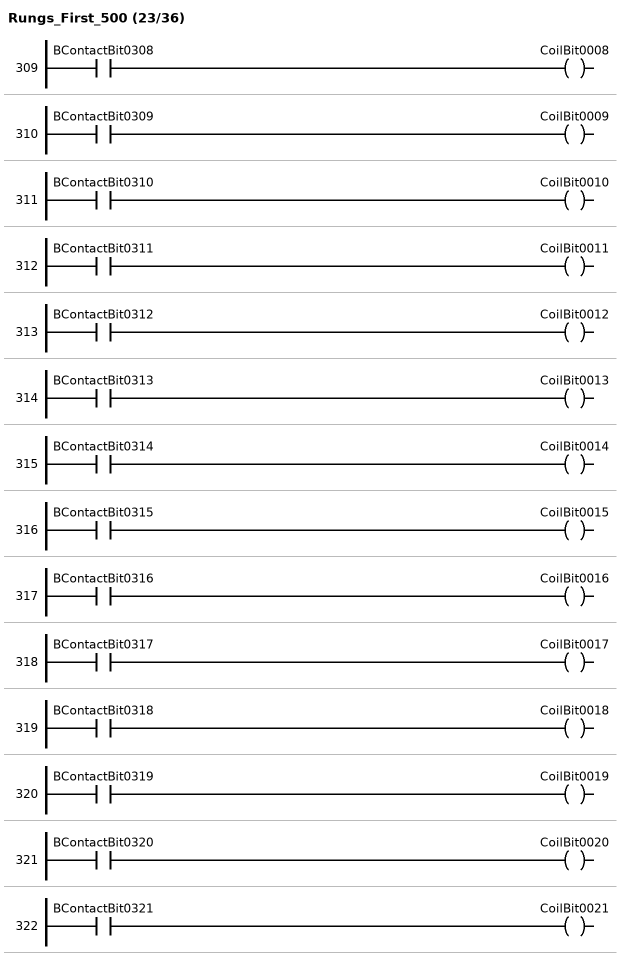
// NETWORK 309
CoilBit0008 := BContactBit0308;

// NETWORK 310
CoilBit0009 := BContactBit0309;

// NETWORK 311
CoilBit0010 := BContactBit0310;

// NETWORK 312
CoilBit0011 := BContactBit0311;

// NETWORK 313
CoilBit0012 := BContactBit0312;

// NETWORK 314
CoilBit0013 := BContactBit0313;

// NETWORK 315
CoilBit0014 := BContactBit0314;

// NETWORK 316
CoilBit0015 := BContactBit0315;

// NETWORK 317
CoilBit0016 := BContactBit0316;

// NETWORK 318
CoilBit0017 := BContactBit0317;

// NETWORK 319
CoilBit0018 := BContactBit0318;

// NETWORK 320
CoilBit0019 := BContactBit0319;

// NETWORK 321
CoilBit0020 := BContactBit0320;

// NETWORK 322
CoilBit0021 := BContactBit0321;

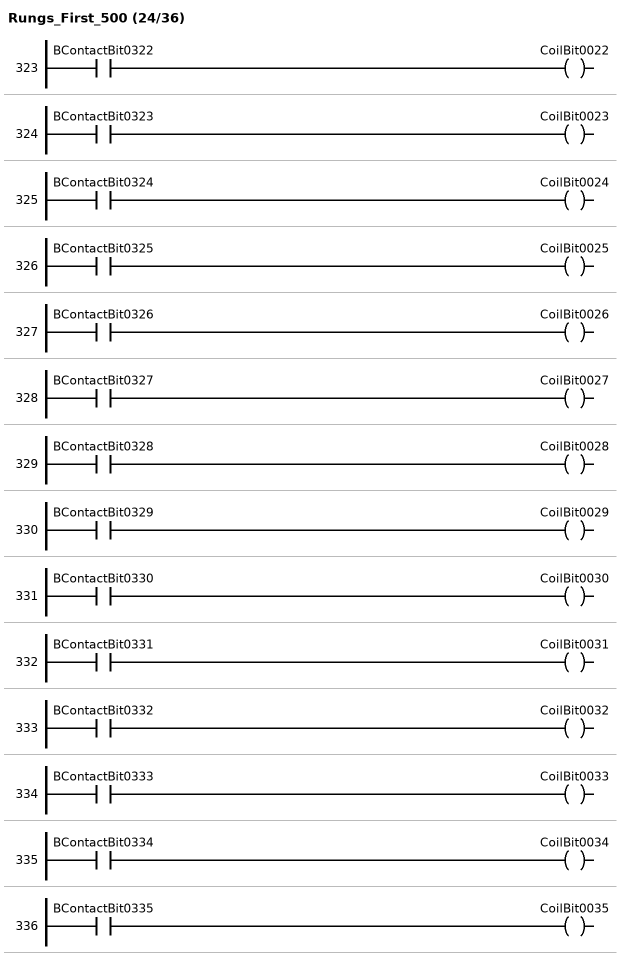
// NETWORK 323
CoilBit0022 := BContactBit0322;

// NETWORK 324
CoilBit0023 := BContactBit0323;

// NETWORK 325
CoilBit0024 := BContactBit0324;

// NETWORK 326
CoilBit0025 := BContactBit0325;

// NETWORK 327
CoilBit0026 := BContactBit0326;

// NETWORK 328
CoilBit0027 := BContactBit0327;

// NETWORK 329
CoilBit0028 := BContactBit0328;

// NETWORK 330
CoilBit0029 := BContactBit0329;

// NETWORK 331
CoilBit0030 := BContactBit0330;

// NETWORK 332
CoilBit0031 := BContactBit0331;

// NETWORK 333
CoilBit0032 := BContactBit0332;

// NETWORK 334
CoilBit0033 := BContactBit0333;

// NETWORK 335
CoilBit0034 := BContactBit0334;

// NETWORK 336
CoilBit0035 := BContactBit0335;

